KUKA KRL program: f1_Kuka_APT204T02S04.SRC

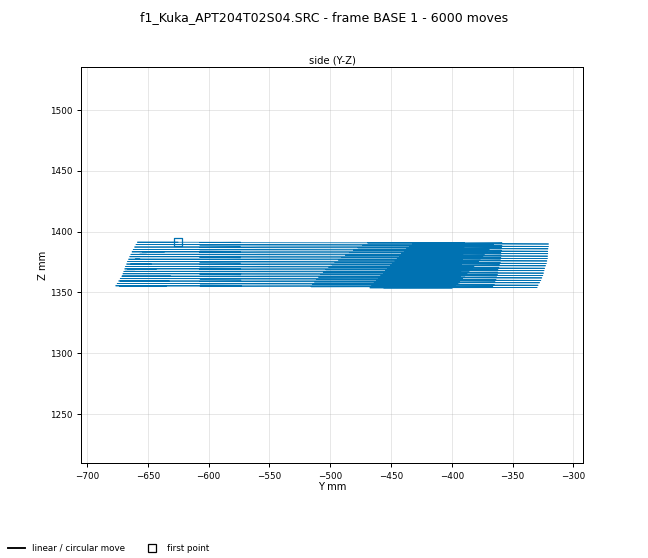
[picture p0: tool path of f1_Kuka_APT204T02S04.SRC in frame BASE 1, 6000 of 6001 moves have a stored position in this frame; points joined in program order, loops and branches not executed]
&ACCESS RVP
&REL 2
&PARAM TEMPLATE = C:\KRC\Roboter\Template\vorgabe
&PARAM EDITMASK = *
DEF f1_Kuka_APT204T02S04()


;FOLD INI;%{PE}%V3.2.0,%MKUKATPBASIS,%CINIT,%VCOMMON,%P
  ;FOLD BAS INI;%{E}%V3.2.0,%MKUKATPBASIS,%CINIT,%VINIT,%P
    GLOBAL INTERRUPT DECL 3 WHEN $STOPMESS==TRUE DO IR_STOPM ( )
    INTERRUPT ON 3
    BAS (#INITMOV,0 )
  ;ENDFOLD (BAS INI)
  ;FOLD USER INI;%{E}%V3.2.0,%MKUKATPUSER,%CINIT,%VINIT,%P
    ;Make your modifications here
  ;ENDFOLD (USER INI)
;ENDFOLD (INI)


;*** Make Null PTP Move
  PTP $pos_act

;*** Auto Load The Correct TOOL Data
  $tool=tool_data[2]

;*** Auto Load The Correct BASE Data
  $base=base_data[1]

  $ADVANCE = 5

;*** Restate Last Velocity
MMPM(30000.0)
SetRPM(8000)
LIN {X -0.143,Y -625.196,Z 1391.416,A 0.000,B 0.000,C 90.000,E1 110.791} C_DIS
LIN {X -0.238,Y -629.866,Z 1391.413,A 0.000,B 0.000,C 90.000,E1 110.301} C_DIS
LIN {X 0.179,Y -634.129,Z 1391.410,A 0.000,B 0.000,C 90.000,E1 109.758} C_DIS
LIN {X 0.021,Y -638.848,Z 1391.406,A 0.000,B 0.000,C 90.000,E1 109.141} C_DIS
LIN {X -0.310,Y -643.103,Z 1391.403,A 0.000,B 0.000,C 90.000,E1 108.544} C_DIS
LIN {X 0.208,Y -646.821,Z 1391.399,A 0.000,B 0.000,C 90.000,E1 107.873} C_DIS
LIN {X -0.083,Y -649.386,Z 1391.397,A 0.000,B 0.000,C 90.000,E1 107.402} C_DIS
LIN {X -0.030,Y -650.571,Z 1391.395,A 0.000,B 0.000,C 90.000,E1 107.149} C_DIS
LIN {X -0.300,Y -652.600,Z 1391.393,A 0.000,B 0.000,C 90.000,E1 106.677} C_DIS
LIN {X 0.197,Y -653.441,Z 1391.391,A 0.000,B 0.000,C 90.000,E1 106.386} C_DIS
LIN {X 0.134,Y -654.835,Z 1391.388,A 0.000,B 0.000,C 90.000,E1 105.898} C_DIS
LIN {X -0.217,Y -656.248,Z 1391.384,A 0.000,B 0.000,C 90.000,E1 105.190} C_DIS
LIN {X 0.139,Y -657.684,Z 1391.379,A 0.000,B 0.000,C 90.000,E1 104.175} C_DIS
LIN {X -0.185,Y -658.387,Z 1391.375,A 0.000,B 0.000,C 90.000,E1 103.467} C_DIS
LIN {X 0.242,Y -658.599,Z 1391.372,A 0.000,B 0.000,C 90.000,E1 102.939} C_DIS
LIN {X -0.216,Y -658.574,Z 1391.368,A 0.000,B 0.000,C 90.000,E1 102.243} C_DIS
LIN {X 0.219,Y -658.347,Z 1391.365,A 0.000,B 0.000,C 90.000,E1 101.715} C_DIS
LIN {X 0.004,Y -657.844,Z 1391.363,A 0.000,B 0.000,C 90.000,E1 101.243} C_DIS
LIN {X -0.340,Y -657.164,Z 1391.360,A 0.000,B 0.000,C 90.000,E1 100.782} C_DIS
LIN {X -0.034,Y -655.750,Z 1391.356,A 0.000,B 0.000,C 90.000,E1 100.018} C_DIS
LIN {X 0.261,Y -654.606,Z 1391.353,A 0.000,B 0.000,C 90.000,E1 99.500} C_DIS
LIN {X 0.012,Y -653.243,Z 1391.350,A 0.000,B 0.000,C 90.000,E1 99.029} C_DIS
LIN {X 0.158,Y -650.750,Z 1391.346,A 0.000,B 0.000,C 90.000,E1 98.276} C_DIS
LIN {X -0.217,Y -648.856,Z 1391.343,A 0.000,B 0.000,C 90.000,E1 97.814} C_DIS
LIN {X -0.196,Y -645.464,Z 1391.339,A 0.000,B 0.000,C 90.000,E1 97.068} C_DIS
LIN {X 0.043,Y -642.991,Z 1391.336,A 0.000,B 0.000,C 90.000,E1 96.549} C_DIS
LIN {X 0.261,Y -640.303,Z 1391.334,A 0.000,B 0.000,C 90.000,E1 96.030} C_DIS
LIN {X 0.262,Y -635.979,Z 1391.329,A 0.000,B 0.000,C 90.000,E1 95.277} C_DIS
LIN {X 0.290,Y -632.062,Z 1391.326,A 0.000,B 0.000,C 90.000,E1 94.645} C_DIS
LIN {X 0.283,Y -627.598,Z 1391.323,A 0.000,B 0.000,C 90.000,E1 94.012} C_DIS
LIN {X -0.280,Y -623.386,Z 1391.320,A 0.000,B 0.000,C 90.000,E1 93.555} C_DIS
LIN {X -0.233,Y -617.142,Z 1391.316,A 0.000,B 0.000,C 90.000,E1 92.922} C_DIS
LIN {X 0.002,Y -609.127,Z 1391.312,A 0.000,B 0.000,C 90.000,E1 92.178} C_DIS
LIN {X -0.133,Y -602.258,Z 1391.309,A 0.000,B 0.000,C 90.000,E1 91.604} C_DIS
LIN {X -0.057,Y -596.480,Z 1391.306,A 0.000,B 0.000,C 90.000,E1 91.146} C_DIS
LIN {X -0.147,Y -589.887,Z 1391.304,A 0.000,B 0.000,C 90.000,E1 90.745} C_DIS
LIN {X -0.112,Y -577.492,Z 1391.301,A 0.000,B 0.000,C 90.000,E1 90.115} C_DIS
LIN {X 0.014,Y -574.202,Z 1391.299,A 0.000,B 0.000,C 90.000,E1 89.771} C_DIS
LIN {X -0.190,Y -573.788,Z 1391.298,A 0.000,B 0.000,C 90.000,E1 89.599} C_DIS
LIN {X -0.045,Y -573.564,Z 1391.296,A 0.000,B 0.000,C 90.000,E1 89.312} C_DIS
LIN {X 0.026,Y -573.965,Z 1391.292,A 0.000,B 0.000,C 90.000,E1 88.625} C_DIS
LIN {X 0.192,Y -575.130,Z 1391.285,A 0.000,B 0.000,C 90.000,E1 87.249} C_DIS
LIN {X -0.193,Y -578.267,Z 1391.267,A 0.000,B 0.000,C 90.000,E1 84.033} C_DIS
LIN {X -0.072,Y -580.429,Z 1391.256,A 0.000,B 0.000,C 90.000,E1 82.129} C_DIS
LIN {X -0.185,Y -582.040,Z 1391.249,A 0.000,B 0.000,C 90.000,E1 80.792} C_DIS
LIN {X -0.262,Y -583.597,Z 1391.241,A 0.000,B 0.000,C 90.000,E1 79.454} C_DIS
LIN {X -0.202,Y -585.007,Z 1391.234,A 0.000,B 0.000,C 90.000,E1 78.105} C_DIS
LIN {X 0.135,Y -586.366,Z 1391.225,A 0.000,B 0.000,C 90.000,E1 76.464} C_DIS
LIN {X -0.014,Y -587.239,Z 1391.219,A 0.000,B 0.000,C 90.000,E1 75.408} C_DIS
LIN {X -0.008,Y -588.007,Z 1391.213,A 0.000,B 0.000,C 90.000,E1 74.338} C_DIS
LIN {X 0.104,Y -588.860,Z 1391.204,A 0.000,B 0.000,C 90.000,E1 72.725} C_DIS
LIN {X -0.146,Y -589.785,Z 1391.195,A 0.000,B 0.000,C 90.000,E1 71.148} C_DIS
LIN {X -0.253,Y -590.554,Z 1391.188,A 0.000,B 0.000,C 90.000,E1 69.826} C_DIS
LIN {X 0.057,Y -591.813,Z 1391.176,A 0.000,B 0.000,C 90.000,E1 67.667} C_DIS
LIN {X 0.193,Y -593.164,Z 1391.166,A 0.000,B 0.000,C 90.000,E1 65.793} C_DIS
LIN {X -0.016,Y -594.849,Z 1391.154,A 0.000,B 0.000,C 90.000,E1 63.691} C_DIS
LIN {X 0.160,Y -595.718,Z 1391.148,A 0.000,B 0.000,C 90.000,E1 62.615} C_DIS
LIN {X -0.128,Y -597.967,Z 1391.133,A 0.000,B 0.000,C 90.000,E1 59.999} C_DIS
LIN {X 0.200,Y -599.678,Z 1391.123,A 0.000,B 0.000,C 90.000,E1 58.122} C_DIS
LIN {X 0.057,Y -601.389,Z 1391.113,A 0.000,B 0.000,C 90.000,E1 56.294} C_DIS
LIN {X -0.219,Y -603.022,Z 1391.103,A 0.000,B 0.000,C 90.000,E1 54.482} C_DIS
LIN {X -0.002,Y -604.422,Z 1391.094,A 0.000,B 0.000,C 90.000,E1 52.889} C_DIS
LIN {X 0.200,Y -605.213,Z 1391.088,A 0.000,B 0.000,C 90.000,E1 51.823} C_DIS
LIN {X -0.070,Y -605.930,Z 1391.082,A 0.000,B 0.000,C 90.000,E1 50.803} C_DIS
LIN {X 0.119,Y -606.746,Z 1391.074,A 0.000,B 0.000,C 90.000,E1 49.218} C_DIS
LIN {X 0.062,Y -607.082,Z 1391.066,A 0.000,B 0.000,C 90.000,E1 47.919} C_DIS
LIN {X 0.003,Y -607.334,Z 1391.059,A 0.000,B 0.000,C 90.000,E1 46.620} C_DIS
LIN {X 0.297,Y -607.326,Z 1391.055,A 0.000,B 0.000,C 90.000,E1 45.810} C_DIS
LIN {X -0.025,Y -607.212,Z 1391.049,A 0.000,B 0.000,C 90.000,E1 44.798} C_DIS
LIN {X -0.096,Y -606.832,Z 1391.042,A 0.000,B 0.000,C 90.000,E1 43.500} C_DIS
LIN {X 0.001,Y -606.333,Z 1391.036,A 0.000,B 0.000,C 90.000,E1 42.447} C_DIS
LIN {X -0.133,Y -605.921,Z 1391.031,A 0.000,B 0.000,C 90.000,E1 41.676} C_DIS
LIN {X -0.214,Y -605.096,Z 1391.024,A 0.000,B 0.000,C 90.000,E1 40.378} C_DIS
LIN {X 0.148,Y -604.051,Z 1391.017,A 0.000,B 0.000,C 90.000,E1 39.036} C_DIS
LIN {X 0.112,Y -602.680,Z 1391.010,A 0.000,B 0.000,C 90.000,E1 37.729} C_DIS
LIN {X 0.030,Y -601.770,Z 1391.005,A 0.000,B 0.000,C 90.000,E1 36.950} C_DIS
LIN {X 0.191,Y -600.161,Z 1391.000,A 0.000,B 0.000,C 90.000,E1 35.884} C_DIS
LIN {X 0.087,Y -598.794,Z 1390.995,A 0.000,B 0.000,C 90.000,E1 35.105} C_DIS
LIN {X -0.033,Y -597.155,Z 1390.991,A 0.000,B 0.000,C 90.000,E1 34.326} C_DIS
LIN {X -0.064,Y -594.161,Z 1390.983,A 0.000,B 0.000,C 90.000,E1 33.007} C_DIS
LIN {X -0.065,Y -592.043,Z 1390.979,A 0.000,B 0.000,C 90.000,E1 32.212} C_DIS
LIN {X -0.080,Y -589.699,Z 1390.974,A 0.000,B 0.000,C 90.000,E1 31.416} C_DIS
LIN {X 0.114,Y -588.884,Z 1390.973,A 0.000,B 0.000,C 90.000,E1 31.131} C_DIS
LIN {X 0.066,Y -586.005,Z 1390.969,A 0.000,B 0.000,C 90.000,E1 30.335} C_DIS
LIN {X -0.011,Y -582.750,Z 1390.964,A 0.000,B 0.000,C 90.000,E1 29.539} C_DIS
LIN {X -0.191,Y -578.488,Z 1390.959,A 0.000,B 0.000,C 90.000,E1 28.615} C_DIS
LIN {X 0.031,Y -575.870,Z 1390.956,A 0.000,B 0.000,C 90.000,E1 28.052} C_DIS
LIN {X -0.003,Y -573.037,Z 1390.953,A 0.000,B 0.000,C 90.000,E1 27.513} C_DIS
LIN {X -0.067,Y -567.662,Z 1390.948,A 0.000,B 0.000,C 90.000,E1 26.565} C_DIS
LIN {X 0.243,Y -563.612,Z 1390.944,A 0.000,B 0.000,C 90.000,E1 25.848} C_DIS
LIN {X -0.139,Y -560.160,Z 1390.941,A 0.000,B 0.000,C 90.000,E1 25.335} C_DIS
LIN {X -0.038,Y -556.507,Z 1390.938,A 0.000,B 0.000,C 90.000,E1 24.771} C_DIS
LIN {X -0.073,Y -551.522,Z 1390.934,A 0.000,B 0.000,C 90.000,E1 24.079} C_DIS
LIN {X 0.085,Y -548.354,Z 1390.931,A 0.000,B 0.000,C 90.000,E1 23.643} C_DIS
LIN {X 0.103,Y -542.913,Z 1390.928,A 0.000,B 0.000,C 90.000,E1 22.950} C_DIS
LIN {X -0.059,Y -537.032,Z 1390.924,A 0.000,B 0.000,C 90.000,E1 22.259} C_DIS
LIN {X -0.231,Y -528.146,Z 1390.918,A 0.000,B 0.000,C 90.000,E1 21.280} C_DIS
LIN {X -0.094,Y -521.657,Z 1390.914,A 0.000,B 0.000,C 90.000,E1 20.556} C_DIS
LIN {X -0.150,Y -512.419,Z 1390.909,A 0.000,B 0.000,C 90.000,E1 19.577} C_DIS
LIN {X -0.058,Y -501.874,Z 1390.903,A 0.000,B 0.000,C 90.000,E1 18.489} C_DIS
LIN {X -0.108,Y -486.810,Z 1390.894,A 0.000,B 0.000,C 90.000,E1 16.968} C_DIS
LIN {X 0.057,Y -471.479,Z 1390.885,A 0.000,B 0.000,C 90.000,E1 15.371} C_DIS
LIN {X -0.025,Y -461.668,Z 1390.880,A 0.000,B 0.000,C 90.000,E1 14.356} C_DIS
LIN {X 0.031,Y -447.810,Z 1390.872,A 0.000,B 0.000,C 90.000,E1 12.883} C_DIS
LIN {X -0.238,Y -428.554,Z 1390.860,A 0.000,B 0.000,C 90.000,E1 10.782} C_DIS
LIN {X -0.101,Y -410.782,Z 1390.848,A 0.000,B 0.000,C 90.000,E1 8.624} C_DIS
LIN {X 0.175,Y -396.943,Z 1390.839,A 0.000,B 0.000,C 90.000,E1 6.891} C_DIS
LIN {X 0.154,Y -392.878,Z 1390.836,A 0.000,B 0.000,C 90.000,E1 6.372} C_DIS
LIN {X 0.048,Y -389.976,Z 1390.833,A 0.000,B 0.000,C 90.000,E1 5.910} C_DIS
LIN {X 0.011,Y -389.942,Z 1390.833,A 0.000,B 0.000,C 90.000,E1 5.910} C_DIS
LIN {X -0.120,Y -389.697,Z 1390.832,A 0.000,B 0.000,C 90.000,E1 5.796} C_DIS
LIN {X -0.158,Y -389.698,Z 1390.832,A 0.000,B 0.000,C 90.000,E1 5.796} C_DIS
LIN {X -0.089,Y -390.823,Z 1390.831,A 0.000,B 0.000,C 90.000,E1 5.625} C_DIS
LIN {X 0.121,Y -393.551,Z 1390.829,A 0.000,B 0.000,C 90.000,E1 5.277} C_DIS
LIN {X 0.038,Y -404.905,Z 1390.824,A 0.000,B 0.000,C 90.000,E1 4.302} C_DIS
LIN {X -0.100,Y -409.448,Z 1390.822,A 0.000,B 0.000,C 90.000,E1 3.898} C_DIS
LIN {X -0.163,Y -412.171,Z 1390.820,A 0.000,B 0.000,C 90.000,E1 3.612} C_DIS
LIN {X -0.101,Y -417.094,Z 1390.817,A 0.000,B 0.000,C 90.000,E1 3.037} C_DIS
LIN {X 0.084,Y -423.352,Z 1390.812,A 0.000,B 0.000,C 90.000,E1 2.178} C_DIS
LIN {X 0.192,Y -427.973,Z 1390.808,A 0.000,B 0.000,C 90.000,E1 1.489} C_DIS
LIN {X -0.107,Y -432.450,Z 1390.805,A 0.000,B 0.000,C 90.000,E1 0.859} C_DIS
LIN {X 0.000,Y -437.845,Z 1390.800,A 0.000,B 0.000,C 90.000,E1 360.000} C_DIS
LIN {X -0.049,Y -443.155,Z 1390.795,A 0.000,B 0.000,C 90.000,E1 359.141} C_DIS
LIN {X 0.209,Y -447.035,Z 1390.792,A 0.000,B 0.000,C 90.000,E1 358.453} C_DIS
LIN {X 0.222,Y -452.233,Z 1390.786,A 0.000,B 0.000,C 90.000,E1 357.478} C_DIS
LIN {X 0.212,Y -456.335,Z 1390.782,A 0.000,B 0.000,C 90.000,E1 356.674} C_DIS
LIN {X 0.118,Y -459.401,Z 1390.778,A 0.000,B 0.000,C 90.000,E1 356.045} C_DIS
LIN {X -0.150,Y -463.497,Z 1390.773,A 0.000,B 0.000,C 90.000,E1 355.122} C_DIS
LIN {X 0.156,Y -465.457,Z 1390.770,A 0.000,B 0.000,C 90.000,E1 354.609} C_DIS
LIN {X 0.156,Y -467.659,Z 1390.767,A 0.000,B 0.000,C 90.000,E1 353.976} C_DIS
LIN {X -0.044,Y -468.494,Z 1390.765,A 0.000,B 0.000,C 90.000,E1 353.685} C_DIS
LIN {X 0.225,Y -469.028,Z 1390.763,A 0.000,B 0.000,C 90.000,E1 353.337} C_DIS
LIN {X -0.023,Y -469.181,Z 1390.761,A 0.000,B 0.000,C 90.000,E1 353.053} C_DIS
LIN {X -0.211,Y -468.449,Z 1390.760,A 0.000,B 0.000,C 90.000,E1 352.761} C_DIS
LIN {X -0.022,Y -467.671,Z 1390.759,A 0.000,B 0.000,C 90.000,E1 352.648} C_DIS
LIN {X -0.135,Y -465.013,Z 1390.759,A 0.000,B 0.000,C 90.000,E1 352.591} C_DIS
LIN {X -0.105,Y -421.785,Z 1390.755,A 0.000,B 0.000,C 90.000,E1 351.837} C_DIS
LIN {X 0.169,Y -384.990,Z 1390.750,A 0.000,B 0.000,C 90.000,E1 351.027} C_DIS
LIN {X 0.119,Y -358.693,Z 1390.747,A 0.000,B 0.000,C 90.000,E1 350.387} C_DIS
LIN {X 0.100,Y -358.666,Z 1390.747,A 0.000,B 0.000,C 90.000,E1 350.387} C_DIS
LIN {X -0.096,Y -359.584,Z 1390.725,A 0.000,B 0.000,C 90.000,E1 346.589} C_DIS
LIN {X -0.088,Y -361.850,Z 1390.684,A 0.000,B 0.000,C 90.000,E1 339.082} C_DIS
LIN {X 0.207,Y -362.253,Z 1390.675,A 0.000,B 0.000,C 90.000,E1 337.539} C_DIS
LIN {X 0.082,Y -366.046,Z 1390.642,A 0.000,B 0.000,C 90.000,E1 331.591} C_DIS
LIN {X -0.212,Y -367.179,Z 1390.630,A 0.000,B 0.000,C 90.000,E1 329.410} C_DIS
LIN {X 0.044,Y -371.805,Z 1390.601,A 0.000,B 0.000,C 90.000,E1 324.196} C_DIS
LIN {X -0.168,Y -377.442,Z 1390.567,A 0.000,B 0.000,C 90.000,E1 318.000} C_DIS
LIN {X 0.112,Y -378.276,Z 1390.563,A 0.000,B 0.000,C 90.000,E1 317.229} C_DIS
LIN {X 0.108,Y -384.028,Z 1390.530,A 0.000,B 0.000,C 90.000,E1 311.434} C_DIS
LIN {X 0.194,Y -384.936,Z 1390.526,A 0.000,B 0.000,C 90.000,E1 310.701} C_DIS
LIN {X -0.177,Y -390.698,Z 1390.495,A 0.000,B 0.000,C 90.000,E1 305.025} C_DIS
LIN {X 0.210,Y -391.195,Z 1390.493,A 0.000,B 0.000,C 90.000,E1 304.612} C_DIS
LIN {X 0.017,Y -396.910,Z 1390.459,A 0.000,B 0.000,C 90.000,E1 298.615} C_DIS
LIN {X -0.109,Y -397.907,Z 1390.449,A 0.000,B 0.000,C 90.000,E1 296.873} C_DIS
LIN {X 0.028,Y -401.639,Z 1390.426,A 0.000,B 0.000,C 90.000,E1 292.642} C_DIS
LIN {X 0.165,Y -404.713,Z 1390.395,A 0.000,B 0.000,C 90.000,E1 287.040} C_DIS
LIN {X 0.168,Y -406.136,Z 1390.364,A 0.000,B 0.000,C 90.000,E1 281.478} C_DIS
LIN {X -0.135,Y -405.443,Z 1390.347,A 0.000,B 0.000,C 90.000,E1 278.398} C_DIS
LIN {X -0.138,Y -405.689,Z 1390.333,A 0.000,B 0.000,C 90.000,E1 275.967} C_DIS
LIN {X -0.067,Y -403.574,Z 1390.306,A 0.000,B 0.000,C 90.000,E1 271.088} C_DIS
LIN {X -0.132,Y -403.240,Z 1390.302,A 0.000,B 0.000,C 90.000,E1 270.401} C_DIS
LIN {X 0.106,Y -399.091,Z 1390.273,A 0.000,B 0.000,C 90.000,E1 265.122} C_DIS
LIN {X 0.048,Y -398.855,Z 1390.271,A 0.000,B 0.000,C 90.000,E1 264.780} C_DIS
LIN {X -0.054,Y -393.336,Z 1390.244,A 0.000,B 0.000,C 90.000,E1 259.859} C_DIS
LIN {X -0.133,Y -392.758,Z 1390.240,A 0.000,B 0.000,C 90.000,E1 259.162} C_DIS
LIN {X -0.054,Y -386.308,Z 1390.214,A 0.000,B 0.000,C 90.000,E1 254.519} C_DIS
LIN {X 0.018,Y -385.205,Z 1390.208,A 0.000,B 0.000,C 90.000,E1 253.433} C_DIS
LIN {X -0.051,Y -383.992,Z 1390.204,A 0.000,B 0.000,C 90.000,E1 252.725} C_DIS
LIN {X -0.221,Y -377.431,Z 1390.180,A 0.000,B 0.000,C 90.000,E1 248.411} C_DIS
LIN {X 0.016,Y -376.161,Z 1390.174,A 0.000,B 0.000,C 90.000,E1 247.283} C_DIS
LIN {X 0.187,Y -368.327,Z 1390.147,A 0.000,B 0.000,C 90.000,E1 242.487} C_DIS
LIN {X -0.097,Y -366.466,Z 1390.139,A 0.000,B 0.000,C 90.000,E1 241.051} C_DIS
LIN {X -0.012,Y -365.918,Z 1390.137,A 0.000,B 0.000,C 90.000,E1 240.667} C_DIS
LIN {X 0.077,Y -359.101,Z 1390.114,A 0.000,B 0.000,C 90.000,E1 236.548} C_DIS
LIN {X 0.164,Y -356.245,Z 1390.102,A 0.000,B 0.000,C 90.000,E1 234.276} C_DIS
LIN {X 0.095,Y -355.717,Z 1390.100,A 0.000,B 0.000,C 90.000,E1 233.909} C_DIS
LIN {X -0.101,Y -348.706,Z 1390.074,A 0.000,B 0.000,C 90.000,E1 229.380} C_DIS
LIN {X -0.027,Y -346.116,Z 1390.062,A 0.000,B 0.000,C 90.000,E1 227.067} C_DIS
LIN {X -0.041,Y -342.667,Z 1390.049,A 0.000,B 0.000,C 90.000,E1 224.757} C_DIS
LIN {X 0.152,Y -336.754,Z 1390.018,A 0.000,B 0.000,C 90.000,E1 219.277} C_DIS
LIN {X 0.062,Y -330.806,Z 1389.988,A 0.000,B 0.000,C 90.000,E1 213.785} C_DIS
LIN {X 0.019,Y -329.252,Z 1389.975,A 0.000,B 0.000,C 90.000,E1 211.416} C_DIS
LIN {X -0.130,Y -324.635,Z 1389.941,A 0.000,B 0.000,C 90.000,E1 205.463} C_DIS
LIN {X 0.062,Y -323.806,Z 1389.928,A 0.000,B 0.000,C 90.000,E1 203.025} C_DIS
LIN {X -0.034,Y -321.131,Z 1389.881,A 0.000,B 0.000,C 90.000,E1 194.592} C_DIS
LIN {X -0.062,Y -320.418,Z 1389.862,A 0.000,B 0.000,C 90.000,E1 191.243} C_DIS
LIN {X -0.092,Y -320.565,Z 1389.862,A 0.000,B 0.000,C 90.000,E1 191.243} C_DIS
LIN {X 0.115,Y -350.932,Z 1389.857,A 0.000,B 0.000,C 90.000,E1 190.254} C_DIS
LIN {X 0.078,Y -384.592,Z 1389.852,A 0.000,B 0.000,C 90.000,E1 189.378} C_DIS
LIN {X 0.108,Y -424.277,Z 1389.847,A 0.000,B 0.000,C 90.000,E1 188.511} C_DIS
LIN {X 0.124,Y -429.421,Z 1389.847,A 0.000,B 0.000,C 90.000,E1 188.398} C_DIS
LIN {X -0.080,Y -430.370,Z 1389.846,A 0.000,B 0.000,C 90.000,E1 188.341} C_DIS
LIN {X 0.070,Y -431.572,Z 1389.845,A 0.000,B 0.000,C 90.000,E1 188.049} C_DIS
LIN {X 0.182,Y -432.160,Z 1389.843,A 0.000,B 0.000,C 90.000,E1 187.701} C_DIS
LIN {X -0.131,Y -432.366,Z 1389.841,A 0.000,B 0.000,C 90.000,E1 187.409} C_DIS
LIN {X 0.051,Y -432.032,Z 1389.837,A 0.000,B 0.000,C 90.000,E1 186.720} C_DIS
LIN {X 0.030,Y -431.325,Z 1389.830,A 0.000,B 0.000,C 90.000,E1 185.391} C_DIS
LIN {X -0.152,Y -430.337,Z 1389.824,A 0.000,B 0.000,C 90.000,E1 184.416} C_DIS
LIN {X 0.018,Y -429.583,Z 1389.821,A 0.000,B 0.000,C 90.000,E1 183.726} C_DIS
LIN {X -0.114,Y -427.646,Z 1389.813,A 0.000,B 0.000,C 90.000,E1 182.407} C_DIS
LIN {X 0.029,Y -426.466,Z 1389.810,A 0.000,B 0.000,C 90.000,E1 181.718} C_DIS
LIN {X 0.205,Y -424.428,Z 1389.804,A 0.000,B 0.000,C 90.000,E1 180.688} C_DIS
LIN {X -0.165,Y -423.680,Z 1389.802,A 0.000,B 0.000,C 90.000,E1 180.401} C_DIS
LIN {X -0.019,Y -420.873,Z 1389.797,A 0.000,B 0.000,C 90.000,E1 179.370} C_DIS
LIN {X 0.057,Y -418.810,Z 1389.793,A 0.000,B 0.000,C 90.000,E1 178.682} C_DIS
LIN {X 0.148,Y -415.012,Z 1389.787,A 0.000,B 0.000,C 90.000,E1 177.650} C_DIS
LIN {X 0.191,Y -411.516,Z 1389.782,A 0.000,B 0.000,C 90.000,E1 176.788} C_DIS
LIN {X 0.190,Y -406.155,Z 1389.777,A 0.000,B 0.000,C 90.000,E1 175.755} C_DIS
LIN {X 0.141,Y -401.143,Z 1389.772,A 0.000,B 0.000,C 90.000,E1 174.894} C_DIS
LIN {X -0.127,Y -387.572,Z 1389.760,A 0.000,B 0.000,C 90.000,E1 172.818} C_DIS
LIN {X -0.015,Y -380.337,Z 1389.753,A 0.000,B 0.000,C 90.000,E1 171.546} C_DIS
LIN {X -0.033,Y -372.669,Z 1389.745,A 0.000,B 0.000,C 90.000,E1 170.095} C_DIS
LIN {X 0.090,Y -369.184,Z 1389.741,A 0.000,B 0.000,C 90.000,E1 169.342} C_DIS
LIN {X 0.017,Y -367.117,Z 1389.738,A 0.000,B 0.000,C 90.000,E1 168.814} C_DIS
LIN {X 0.005,Y -365.770,Z 1389.735,A 0.000,B 0.000,C 90.000,E1 168.285} C_DIS
LIN {X -0.032,Y -365.767,Z 1389.735,A 0.000,B 0.000,C 90.000,E1 168.285} C_DIS
LIN {X 0.093,Y -366.445,Z 1389.733,A 0.000,B 0.000,C 90.000,E1 167.825} C_DIS
LIN {X 0.056,Y -366.477,Z 1389.732,A 0.000,B 0.000,C 90.000,E1 167.825} C_DIS
LIN {X -0.040,Y -369.073,Z 1389.730,A 0.000,B 0.000,C 90.000,E1 167.353} C_DIS
LIN {X 0.057,Y -376.139,Z 1389.725,A 0.000,B 0.000,C 90.000,E1 166.408} C_DIS
LIN {X -0.008,Y -383.314,Z 1389.720,A 0.000,B 0.000,C 90.000,E1 165.589} C_DIS
LIN {X -0.071,Y -395.482,Z 1389.713,A 0.000,B 0.000,C 90.000,E1 164.338} C_DIS
LIN {X 0.143,Y -407.819,Z 1389.707,A 0.000,B 0.000,C 90.000,E1 163.142} C_DIS
LIN {X -0.231,Y -431.267,Z 1389.696,A 0.000,B 0.000,C 90.000,E1 161.221} C_DIS
LIN {X 0.064,Y -443.907,Z 1389.690,A 0.000,B 0.000,C 90.000,E1 160.188} C_DIS
LIN {X -0.031,Y -454.875,Z 1389.685,A 0.000,B 0.000,C 90.000,E1 159.337} C_DIS
LIN {X -0.012,Y -465.637,Z 1389.680,A 0.000,B 0.000,C 90.000,E1 158.465} C_DIS
LIN {X -0.180,Y -473.094,Z 1389.677,A 0.000,B 0.000,C 90.000,E1 157.847} C_DIS
LIN {X -0.046,Y -478.923,Z 1389.674,A 0.000,B 0.000,C 90.000,E1 157.305} C_DIS
LIN {X -0.136,Y -487.315,Z 1389.670,A 0.000,B 0.000,C 90.000,E1 156.538} C_DIS
LIN {X -0.108,Y -494.325,Z 1389.666,A 0.000,B 0.000,C 90.000,E1 155.869} C_DIS
LIN {X -0.040,Y -502.435,Z 1389.661,A 0.000,B 0.000,C 90.000,E1 155.025} C_DIS
LIN {X -0.105,Y -507.695,Z 1389.658,A 0.000,B 0.000,C 90.000,E1 154.460} C_DIS
LIN {X -0.048,Y -514.044,Z 1389.654,A 0.000,B 0.000,C 90.000,E1 153.717} C_DIS
LIN {X -0.213,Y -519.975,Z 1389.650,A 0.000,B 0.000,C 90.000,E1 152.999} C_DIS
LIN {X -0.005,Y -523.355,Z 1389.647,A 0.000,B 0.000,C 90.000,E1 152.538} C_DIS
LIN {X -0.022,Y -526.518,Z 1389.645,A 0.000,B 0.000,C 90.000,E1 152.103} C_DIS
LIN {X 0.074,Y -530.265,Z 1389.642,A 0.000,B 0.000,C 90.000,E1 151.513} C_DIS
LIN {X 0.055,Y -534.335,Z 1389.638,A 0.000,B 0.000,C 90.000,E1 150.795} C_DIS
LIN {X 0.210,Y -537.186,Z 1389.635,A 0.000,B 0.000,C 90.000,E1 150.205} C_DIS
LIN {X -0.220,Y -540.124,Z 1389.631,A 0.000,B 0.000,C 90.000,E1 149.537} C_DIS
LIN {X -0.028,Y -542.270,Z 1389.628,A 0.000,B 0.000,C 90.000,E1 148.948} C_DIS
LIN {X 0.195,Y -545.040,Z 1389.623,A 0.000,B 0.000,C 90.000,E1 148.074} C_DIS
LIN {X -0.041,Y -546.655,Z 1389.620,A 0.000,B 0.000,C 90.000,E1 147.533} C_DIS
LIN {X -0.230,Y -548.631,Z 1389.615,A 0.000,B 0.000,C 90.000,E1 146.707} C_DIS
LIN {X 0.368,Y -550.363,Z 1389.610,A 0.000,B 0.000,C 90.000,E1 145.801} C_DIS
LIN {X 0.222,Y -551.768,Z 1389.606,A 0.000,B 0.000,C 90.000,E1 144.975} C_DIS
LIN {X 0.086,Y -552.876,Z 1389.601,A 0.000,B 0.000,C 90.000,E1 144.149} C_DIS
LIN {X -0.094,Y -553.976,Z 1389.595,A 0.000,B 0.000,C 90.000,E1 143.050} C_DIS
LIN {X -0.097,Y -555.317,Z 1389.585,A 0.000,B 0.000,C 90.000,E1 141.376} C_DIS
LIN {X -0.155,Y -556.399,Z 1389.578,A 0.000,B 0.000,C 90.000,E1 139.989} C_DIS
LIN {X 0.007,Y -556.905,Z 1389.573,A 0.000,B 0.000,C 90.000,E1 139.138} C_DIS
LIN {X -0.088,Y -557.589,Z 1389.565,A 0.000,B 0.000,C 90.000,E1 137.757} C_DIS
LIN {X -0.065,Y -558.334,Z 1389.555,A 0.000,B 0.000,C 90.000,E1 135.810} C_DIS
LIN {X -0.162,Y -558.860,Z 1389.547,A 0.000,B 0.000,C 90.000,E1 134.433} C_DIS
LIN {X -0.183,Y -559.391,Z 1389.538,A 0.000,B 0.000,C 90.000,E1 132.771} C_DIS
LIN {X 0.214,Y -559.667,Z 1389.528,A 0.000,B 0.000,C 90.000,E1 131.067} C_DIS
LIN {X -0.022,Y -560.050,Z 1389.518,A 0.000,B 0.000,C 90.000,E1 129.152} C_DIS
LIN {X -0.243,Y -560.611,Z 1389.507,A 0.000,B 0.000,C 90.000,E1 127.237} C_DIS
LIN {X 0.238,Y -561.334,Z 1389.499,A 0.000,B 0.000,C 90.000,E1 125.804} C_DIS
LIN {X -0.005,Y -561.741,Z 1389.497,A 0.000,B 0.000,C 90.000,E1 125.518} C_DIS
LIN {X -0.352,Y -562.723,Z 1389.496,A 0.000,B 0.000,C 90.000,E1 125.311} C_DIS
LIN {X 0.082,Y -563.387,Z 1389.494,A 0.000,B 0.000,C 90.000,E1 124.978} C_DIS
LIN {X 0.039,Y -563.430,Z 1389.494,A 0.000,B 0.000,C 90.000,E1 124.978} C_DIS
LIN {X -0.041,Y -565.054,Z 1389.494,A 0.000,B 0.000,C 90.000,E1 124.865} C_DIS
LIN {X -0.259,Y -566.721,Z 1389.493,A 0.000,B 0.000,C 90.000,E1 124.818} C_DIS
LIN {X -0.196,Y -570.932,Z 1389.493,A 0.000,B 0.000,C 90.000,E1 124.692} C_DIS
LIN {X 0.099,Y -576.932,Z 1389.492,A 0.000,B 0.000,C 90.000,E1 124.532} C_DIS
LIN {X 0.090,Y -583.270,Z 1389.491,A 0.000,B 0.000,C 90.000,E1 124.358} C_DIS
LIN {X 0.074,Y -588.758,Z 1389.490,A 0.000,B 0.000,C 90.000,E1 124.119} C_DIS
LIN {X 0.168,Y -594.673,Z 1389.488,A 0.000,B 0.000,C 90.000,E1 123.785} C_DIS
LIN {X 0.059,Y -600.403,Z 1389.486,A 0.000,B 0.000,C 90.000,E1 123.420} C_DIS
LIN {X -0.015,Y -605.851,Z 1389.483,A 0.000,B 0.000,C 90.000,E1 123.007} C_DIS
LIN {X 0.199,Y -612.491,Z 1389.480,A 0.000,B 0.000,C 90.000,E1 122.418} C_DIS
LIN {X -0.116,Y -615.103,Z 1389.479,A 0.000,B 0.000,C 90.000,E1 122.212} C_DIS
LIN {X -0.069,Y -620.916,Z 1389.476,A 0.000,B 0.000,C 90.000,E1 121.592} C_DIS
LIN {X -0.090,Y -624.377,Z 1389.473,A 0.000,B 0.000,C 90.000,E1 121.209} C_DIS
LIN {X -0.285,Y -631.549,Z 1389.468,A 0.000,B 0.000,C 90.000,E1 120.335} C_DIS
LIN {X 0.105,Y -635.824,Z 1389.465,A 0.000,B 0.000,C 90.000,E1 119.667} C_DIS
LIN {X 0.195,Y -639.048,Z 1389.462,A 0.000,B 0.000,C 90.000,E1 119.155} C_DIS
LIN {X -0.220,Y -642.382,Z 1389.459,A 0.000,B 0.000,C 90.000,E1 118.565} C_DIS
LIN {X 0.152,Y -643.495,Z 1389.457,A 0.000,B 0.000,C 90.000,E1 118.281} C_DIS
LIN {X 0.294,Y -645.428,Z 1389.454,A 0.000,B 0.000,C 90.000,E1 117.769} C_DIS
LIN {X 0.371,Y -646.208,Z 1389.453,A 0.000,B 0.000,C 90.000,E1 117.513} C_DIS
LIN {X -0.041,Y -647.245,Z 1389.450,A 0.000,B 0.000,C 90.000,E1 117.052} C_DIS
LIN {X 0.043,Y -647.666,Z 1389.449,A 0.000,B 0.000,C 90.000,E1 116.796} C_DIS
LIN {X 0.129,Y -647.863,Z 1389.448,A 0.000,B 0.000,C 90.000,E1 116.539} C_DIS
LIN {X -0.072,Y -647.895,Z 1389.446,A 0.000,B 0.000,C 90.000,E1 116.309} C_DIS
LIN {X 0.198,Y -647.461,Z 1389.442,A 0.000,B 0.000,C 90.000,E1 115.540} C_DIS
LIN {X -0.212,Y -646.859,Z 1389.439,A 0.000,B 0.000,C 90.000,E1 115.079} C_DIS
LIN {X -0.128,Y -646.078,Z 1389.438,A 0.000,B 0.000,C 90.000,E1 114.823} C_DIS
LIN {X -0.232,Y -644.029,Z 1389.435,A 0.000,B 0.000,C 90.000,E1 114.335} C_DIS
LIN {X -0.084,Y -640.444,Z 1389.432,A 0.000,B 0.000,C 90.000,E1 113.823} C_DIS
LIN {X -0.053,Y -639.110,Z 1389.432,A 0.000,B 0.000,C 90.000,E1 113.695} C_DIS
LIN {X 0.212,Y -635.318,Z 1389.431,A 0.000,B 0.000,C 90.000,E1 113.462} C_DIS
LIN {X 0.116,Y -634.024,Z 1389.430,A 0.000,B 0.000,C 90.000,E1 113.387} C_DIS
LIN {X 0.270,Y -632.549,Z 1389.429,A 0.000,B 0.000,C 90.000,E1 113.259} C_DIS
LIN {X -0.344,Y -630.253,Z 1389.429,A 0.000,B 0.000,C 90.000,E1 113.206} C_DIS
LIN {X -0.112,Y -628.422,Z 1389.428,A 0.000,B 0.000,C 90.000,E1 113.131} C_DIS
LIN {X 0.252,Y -623.334,Z 1389.427,A 0.000,B 0.000,C 90.000,E1 112.898} C_DIS
LIN {X 0.292,Y -621.466,Z 1389.427,A 0.000,B 0.000,C 90.000,E1 112.823} C_DIS
LIN {X -0.010,Y -608.882,Z 1389.425,A 0.000,B 0.000,C 90.000,E1 112.461} C_DIS
LIN {X -0.043,Y -608.884,Z 1389.425,A 0.000,B 0.000,C 90.000,E1 112.461} C_DIS
LIN {X 0.139,Y -611.746,Z 1389.423,A 0.000,B 0.000,C 90.000,E1 112.153} C_DIS
LIN {X 0.064,Y -614.838,Z 1389.422,A 0.000,B 0.000,C 90.000,E1 111.897} C_DIS
LIN {X 0.306,Y -621.292,Z 1389.418,A 0.000,B 0.000,C 90.000,E1 111.280} C_DIS
LIN {X -0.243,Y -625.045,Z 1389.416,A 0.000,B 0.000,C 90.000,E1 110.972} C_DIS
LIN {X 0.285,Y -629.756,Z 1389.414,A 0.000,B 0.000,C 90.000,E1 110.429} C_DIS
LIN {X 0.113,Y -635.026,Z 1389.410,A 0.000,B 0.000,C 90.000,E1 109.812} C_DIS
LIN {X -0.249,Y -639.706,Z 1389.407,A 0.000,B 0.000,C 90.000,E1 109.214} C_DIS
LIN {X 0.243,Y -643.906,Z 1389.403,A 0.000,B 0.000,C 90.000,E1 108.544} C_DIS
LIN {X -0.042,Y -647.643,Z 1389.400,A 0.000,B 0.000,C 90.000,E1 107.946} C_DIS
LIN {X -0.104,Y -650.825,Z 1389.396,A 0.000,B 0.000,C 90.000,E1 107.330} C_DIS
LIN {X 0.126,Y -653.948,Z 1389.392,A 0.000,B 0.000,C 90.000,E1 106.567} C_DIS
LIN {X -0.050,Y -656.073,Z 1389.388,A 0.000,B 0.000,C 90.000,E1 105.843} C_DIS
LIN {X -0.388,Y -657.439,Z 1389.384,A 0.000,B 0.000,C 90.000,E1 105.134} C_DIS
LIN {X -0.013,Y -658.898,Z 1389.379,A 0.000,B 0.000,C 90.000,E1 104.120} C_DIS
LIN {X 0.316,Y -659.550,Z 1389.374,A 0.000,B 0.000,C 90.000,E1 103.355} C_DIS
LIN {X 0.113,Y -659.765,Z 1389.372,A 0.000,B 0.000,C 90.000,E1 102.883} C_DIS
LIN {X -0.193,Y -659.677,Z 1389.368,A 0.000,B 0.000,C 90.000,E1 102.175} C_DIS
LIN {X 0.111,Y -659.420,Z 1389.365,A 0.000,B 0.000,C 90.000,E1 101.658} C_DIS
LIN {X -0.096,Y -658.910,Z 1389.362,A 0.000,B 0.000,C 90.000,E1 101.186} C_DIS
LIN {X 0.338,Y -658.236,Z 1389.359,A 0.000,B 0.000,C 90.000,E1 100.658} C_DIS
LIN {X -0.114,Y -656.751,Z 1389.355,A 0.000,B 0.000,C 90.000,E1 99.962} C_DIS
LIN {X 0.190,Y -655.575,Z 1389.353,A 0.000,B 0.000,C 90.000,E1 99.443} C_DIS
LIN {X -0.052,Y -654.185,Z 1389.350,A 0.000,B 0.000,C 90.000,E1 98.973} C_DIS
LIN {X 0.239,Y -652.557,Z 1389.347,A 0.000,B 0.000,C 90.000,E1 98.454} C_DIS
LIN {X -0.124,Y -650.743,Z 1389.344,A 0.000,B 0.000,C 90.000,E1 97.992} C_DIS
LIN {X 0.001,Y -647.508,Z 1389.340,A 0.000,B 0.000,C 90.000,E1 97.239} C_DIS
LIN {X 0.132,Y -644.442,Z 1389.337,A 0.000,B 0.000,C 90.000,E1 96.606} C_DIS
LIN {X 0.305,Y -641.109,Z 1389.333,A 0.000,B 0.000,C 90.000,E1 95.967} C_DIS
LIN {X 0.247,Y -636.768,Z 1389.329,A 0.000,B 0.000,C 90.000,E1 95.220} C_DIS
LIN {X 0.282,Y -632.828,Z 1389.326,A 0.000,B 0.000,C 90.000,E1 94.588} C_DIS
LIN {X -0.254,Y -629.328,Z 1389.323,A 0.000,B 0.000,C 90.000,E1 94.131} C_DIS
LIN {X -0.277,Y -624.144,Z 1389.319,A 0.000,B 0.000,C 90.000,E1 93.498} C_DIS
LIN {X -0.225,Y -617.887,Z 1389.316,A 0.000,B 0.000,C 90.000,E1 92.865} C_DIS
LIN {X -0.013,Y -609.915,Z 1389.312,A 0.000,B 0.000,C 90.000,E1 92.121} C_DIS
LIN {X -0.165,Y -603.071,Z 1389.309,A 0.000,B 0.000,C 90.000,E1 91.547} C_DIS
LIN {X -0.131,Y -597.199,Z 1389.306,A 0.000,B 0.000,C 90.000,E1 91.088} C_DIS
LIN {X -0.177,Y -590.715,Z 1389.304,A 0.000,B 0.000,C 90.000,E1 90.688} C_DIS
LIN {X -0.037,Y -585.411,Z 1389.302,A 0.000,B 0.000,C 90.000,E1 90.401} C_DIS
LIN {X -0.277,Y -577.995,Z 1389.300,A 0.000,B 0.000,C 90.000,E1 90.057} C_DIS
LIN {X -0.113,Y -577.349,Z 1389.300,A 0.000,B 0.000,C 90.000,E1 90.000} C_DIS
LIN {X 0.279,Y -574.336,Z 1389.298,A 0.000,B 0.000,C 90.000,E1 89.656} C_DIS
LIN {X 0.238,Y -574.303,Z 1389.298,A 0.000,B 0.000,C 90.000,E1 89.656} C_DIS
LIN {X 0.008,Y -573.679,Z 1389.297,A 0.000,B 0.000,C 90.000,E1 89.427} C_DIS
LIN {X -0.098,Y -573.665,Z 1389.295,A 0.000,B 0.000,C 90.000,E1 89.026} C_DIS
LIN {X -0.220,Y -575.204,Z 1389.284,A 0.000,B 0.000,C 90.000,E1 87.135} C_DIS
LIN {X -0.177,Y -578.062,Z 1389.267,A 0.000,B 0.000,C 90.000,E1 84.147} C_DIS
LIN {X -0.057,Y -580.243,Z 1389.257,A 0.000,B 0.000,C 90.000,E1 82.243} C_DIS
LIN {X -0.034,Y -582.170,Z 1389.248,A 0.000,B 0.000,C 90.000,E1 80.622} C_DIS
LIN {X -0.116,Y -583.737,Z 1389.240,A 0.000,B 0.000,C 90.000,E1 79.285} C_DIS
LIN {X 0.270,Y -584.824,Z 1389.234,A 0.000,B 0.000,C 90.000,E1 78.173} C_DIS
LIN {X 0.023,Y -586.236,Z 1389.226,A 0.000,B 0.000,C 90.000,E1 76.589} C_DIS
LIN {X 0.013,Y -587.119,Z 1389.220,A 0.000,B 0.000,C 90.000,E1 75.519} C_DIS
LIN {X 0.271,Y -588.039,Z 1389.212,A 0.000,B 0.000,C 90.000,E1 74.157} C_DIS
LIN {X -0.177,Y -588.918,Z 1389.203,A 0.000,B 0.000,C 90.000,E1 72.598} C_DIS
LIN {X -0.184,Y -590.005,Z 1389.193,A 0.000,B 0.000,C 90.000,E1 70.732} C_DIS
LIN {X 0.029,Y -590.597,Z 1389.187,A 0.000,B 0.000,C 90.000,E1 69.645} C_DIS
LIN {X -0.100,Y -591.689,Z 1389.177,A 0.000,B 0.000,C 90.000,E1 67.794} C_DIS
LIN {X 0.030,Y -593.013,Z 1389.166,A 0.000,B 0.000,C 90.000,E1 65.921} C_DIS
LIN {X -0.003,Y -594.282,Z 1389.157,A 0.000,B 0.000,C 90.000,E1 64.332} C_DIS
LIN {X -0.009,Y -595.621,Z 1389.149,A 0.000,B 0.000,C 90.000,E1 62.743} C_DIS
LIN {X 0.219,Y -597.840,Z 1389.134,A 0.000,B 0.000,C 90.000,E1 60.078} C_DIS
LIN {X 0.027,Y -599.569,Z 1389.124,A 0.000,B 0.000,C 90.000,E1 58.250} C_DIS
LIN {X -0.355,Y -600.997,Z 1389.115,A 0.000,B 0.000,C 90.000,E1 56.707} C_DIS
LIN {X -0.301,Y -602.183,Z 1389.108,A 0.000,B 0.000,C 90.000,E1 55.388} C_DIS
LIN {X -0.229,Y -603.400,Z 1389.100,A 0.000,B 0.000,C 90.000,E1 54.069} C_DIS
LIN {X -0.008,Y -604.763,Z 1389.092,A 0.000,B 0.000,C 90.000,E1 52.477} C_DIS
LIN {X -0.020,Y -605.696,Z 1389.084,A 0.000,B 0.000,C 90.000,E1 51.170} C_DIS
LIN {X 0.100,Y -606.288,Z 1389.078,A 0.000,B 0.000,C 90.000,E1 50.114} C_DIS
LIN {X -0.164,Y -606.803,Z 1389.073,A 0.000,B 0.000,C 90.000,E1 49.094} C_DIS
LIN {X -0.294,Y -607.031,Z 1389.068,A 0.000,B 0.000,C 90.000,E1 48.324} C_DIS
LIN {X -0.131,Y -607.333,Z 1389.060,A 0.000,B 0.000,C 90.000,E1 46.743} C_DIS
LIN {X -0.008,Y -607.319,Z 1389.054,A 0.000,B 0.000,C 90.000,E1 45.688} C_DIS
LIN {X -0.333,Y -607.213,Z 1389.048,A 0.000,B 0.000,C 90.000,E1 44.676} C_DIS
LIN {X -0.228,Y -606.882,Z 1389.042,A 0.000,B 0.000,C 90.000,E1 43.623} C_DIS
LIN {X 0.311,Y -606.452,Z 1389.036,A 0.000,B 0.000,C 90.000,E1 42.528} C_DIS
LIN {X 0.042,Y -605.555,Z 1389.028,A 0.000,B 0.000,C 90.000,E1 40.987} C_DIS
LIN {X 0.156,Y -604.828,Z 1389.022,A 0.000,B 0.000,C 90.000,E1 39.930} C_DIS
LIN {X -0.126,Y -603.989,Z 1389.016,A 0.000,B 0.000,C 90.000,E1 38.910} C_DIS
LIN {X -0.156,Y -602.662,Z 1389.009,A 0.000,B 0.000,C 90.000,E1 37.604} C_DIS
LIN {X 0.020,Y -601.253,Z 1389.003,A 0.000,B 0.000,C 90.000,E1 36.537} C_DIS
LIN {X -0.311,Y -599.615,Z 1388.997,A 0.000,B 0.000,C 90.000,E1 35.518} C_DIS
LIN {X 0.069,Y -598.112,Z 1388.993,A 0.000,B 0.000,C 90.000,E1 34.692} C_DIS
LIN {X 0.167,Y -595.792,Z 1388.987,A 0.000,B 0.000,C 90.000,E1 33.627} C_DIS
LIN {X 0.179,Y -593.891,Z 1388.983,A 0.000,B 0.000,C 90.000,E1 32.832} C_DIS
LIN {X -0.115,Y -591.058,Z 1388.977,A 0.000,B 0.000,C 90.000,E1 31.799} C_DIS
LIN {X -0.028,Y -589.418,Z 1388.974,A 0.000,B 0.000,C 90.000,E1 31.258} C_DIS
LIN {X -0.071,Y -586.592,Z 1388.969,A 0.000,B 0.000,C 90.000,E1 30.463} C_DIS
LIN {X -0.018,Y -584.540,Z 1388.966,A 0.000,B 0.000,C 90.000,E1 29.922} C_DIS
LIN {X -0.269,Y -582.304,Z 1388.963,A 0.000,B 0.000,C 90.000,E1 29.411} C_DIS
LIN {X 0.055,Y -577.973,Z 1388.958,A 0.000,B 0.000,C 90.000,E1 28.437} C_DIS
LIN {X 0.036,Y -575.283,Z 1388.955,A 0.000,B 0.000,C 90.000,E1 27.897} C_DIS
LIN {X -0.271,Y -572.388,Z 1388.952,A 0.000,B 0.000,C 90.000,E1 27.385} C_DIS
LIN {X 0.000,Y -567.763,Z 1388.948,A 0.000,B 0.000,C 90.000,E1 26.539} C_DIS
LIN {X 0.060,Y -563.699,Z 1388.944,A 0.000,B 0.000,C 90.000,E1 25.848} C_DIS
LIN {X 0.186,Y -560.240,Z 1388.941,A 0.000,B 0.000,C 90.000,E1 25.283} C_DIS
LIN {X -0.218,Y -556.579,Z 1388.938,A 0.000,B 0.000,C 90.000,E1 24.771} C_DIS
LIN {X -0.140,Y -552.658,Z 1388.934,A 0.000,B 0.000,C 90.000,E1 24.207} C_DIS
LIN {X 0.025,Y -549.591,Z 1388.932,A 0.000,B 0.000,C 90.000,E1 23.770} C_DIS
LIN {X -0.135,Y -541.907,Z 1388.927,A 0.000,B 0.000,C 90.000,E1 22.823} C_DIS
LIN {X 0.191,Y -535.944,Z 1388.923,A 0.000,B 0.000,C 90.000,E1 22.078} C_DIS
LIN {X -0.101,Y -525.734,Z 1388.917,A 0.000,B 0.000,C 90.000,E1 20.972} C_DIS
LIN {X 0.150,Y -520.447,Z 1388.913,A 0.000,B 0.000,C 90.000,E1 20.375} C_DIS
LIN {X -0.178,Y -512.630,Z 1388.909,A 0.000,B 0.000,C 90.000,E1 19.577} C_DIS
LIN {X 0.233,Y -501.731,Z 1388.902,A 0.000,B 0.000,C 90.000,E1 18.417} C_DIS
LIN {X 0.096,Y -485.679,Z 1388.893,A 0.000,B 0.000,C 90.000,E1 16.804} C_DIS
LIN {X -0.257,Y -469.071,Z 1388.884,A 0.000,B 0.000,C 90.000,E1 15.134} C_DIS
LIN {X -0.113,Y -460.631,Z 1388.879,A 0.000,B 0.000,C 90.000,E1 14.245} C_DIS
LIN {X -0.169,Y -448.185,Z 1388.872,A 0.000,B 0.000,C 90.000,E1 12.939} C_DIS
LIN {X -0.067,Y -428.748,Z 1388.860,A 0.000,B 0.000,C 90.000,E1 10.782} C_DIS
LIN {X 0.060,Y -412.336,Z 1388.849,A 0.000,B 0.000,C 90.000,E1 8.803} C_DIS
LIN {X 0.101,Y -399.988,Z 1388.841,A 0.000,B 0.000,C 90.000,E1 7.296} C_DIS
LIN {X 0.145,Y -393.201,Z 1388.836,A 0.000,B 0.000,C 90.000,E1 6.429} C_DIS
LIN {X 0.071,Y -390.996,Z 1388.834,A 0.000,B 0.000,C 90.000,E1 6.087} C_DIS
LIN {X 0.142,Y -390.045,Z 1388.833,A 0.000,B 0.000,C 90.000,E1 5.910} C_DIS
LIN {X 0.104,Y -390.019,Z 1388.833,A 0.000,B 0.000,C 90.000,E1 5.910} C_DIS
LIN {X 0.152,Y -389.954,Z 1388.833,A 0.000,B 0.000,C 90.000,E1 5.853} C_DIS
LIN {X 0.115,Y -389.982,Z 1388.833,A 0.000,B 0.000,C 90.000,E1 5.853} C_DIS
LIN {X -0.026,Y -392.093,Z 1388.831,A 0.000,B 0.000,C 90.000,E1 5.568} C_DIS
LIN {X -0.037,Y -393.632,Z 1388.830,A 0.000,B 0.000,C 90.000,E1 5.391} C_DIS
LIN {X 0.080,Y -405.433,Z 1388.824,A 0.000,B 0.000,C 90.000,E1 4.359} C_DIS
LIN {X 0.188,Y -411.425,Z 1388.821,A 0.000,B 0.000,C 90.000,E1 3.784} C_DIS
LIN {X -0.035,Y -418.211,Z 1388.817,A 0.000,B 0.000,C 90.000,E1 3.037} C_DIS
LIN {X -0.005,Y -424.242,Z 1388.813,A 0.000,B 0.000,C 90.000,E1 2.236} C_DIS
LIN {X 0.156,Y -428.867,Z 1388.809,A 0.000,B 0.000,C 90.000,E1 1.547} C_DIS
LIN {X -0.095,Y -434.471,Z 1388.804,A 0.000,B 0.000,C 90.000,E1 0.745} C_DIS
LIN {X 0.167,Y -440.466,Z 1388.799,A 0.000,B 0.000,C 90.000,E1 359.771} C_DIS
LIN {X -0.039,Y -444.537,Z 1388.795,A 0.000,B 0.000,C 90.000,E1 359.141} C_DIS
LIN {X -0.217,Y -448.419,Z 1388.792,A 0.000,B 0.000,C 90.000,E1 358.511} C_DIS
LIN {X -0.193,Y -453.652,Z 1388.786,A 0.000,B 0.000,C 90.000,E1 357.535} C_DIS
LIN {X -0.192,Y -457.755,Z 1388.782,A 0.000,B 0.000,C 90.000,E1 356.731} C_DIS
LIN {X 0.182,Y -460.821,Z 1388.778,A 0.000,B 0.000,C 90.000,E1 356.045} C_DIS
LIN {X -0.069,Y -464.979,Z 1388.773,A 0.000,B 0.000,C 90.000,E1 355.122} C_DIS
LIN {X -0.205,Y -469.456,Z 1388.767,A 0.000,B 0.000,C 90.000,E1 354.033} C_DIS
LIN {X 0.068,Y -470.614,Z 1388.765,A 0.000,B 0.000,C 90.000,E1 353.685} C_DIS
LIN {X -0.122,Y -471.611,Z 1388.763,A 0.000,B 0.000,C 90.000,E1 353.394} C_DIS
LIN {X 0.106,Y -472.464,Z 1388.761,A 0.000,B 0.000,C 90.000,E1 353.053} C_DIS
LIN {X -0.075,Y -473.054,Z 1388.760,A 0.000,B 0.000,C 90.000,E1 352.761} C_DIS
LIN {X 0.218,Y -473.333,Z 1388.758,A 0.000,B 0.000,C 90.000,E1 352.413} C_DIS
LIN {X -0.019,Y -473.013,Z 1388.756,A 0.000,B 0.000,C 90.000,E1 352.129} C_DIS
LIN {X 0.162,Y -472.275,Z 1388.755,A 0.000,B 0.000,C 90.000,E1 351.951} C_DIS
LIN {X -0.014,Y -471.306,Z 1388.755,A 0.000,B 0.000,C 90.000,E1 351.894} C_DIS
LIN {X 0.114,Y -456.133,Z 1388.753,A 0.000,B 0.000,C 90.000,E1 351.602} C_DIS
LIN {X 0.153,Y -415.789,Z 1388.749,A 0.000,B 0.000,C 90.000,E1 350.792} C_DIS
LIN {X 0.157,Y -379.662,Z 1388.744,A 0.000,B 0.000,C 90.000,E1 349.926} C_DIS
LIN {X -0.151,Y -358.859,Z 1388.741,A 0.000,B 0.000,C 90.000,E1 349.398} C_DIS
LIN {X -0.171,Y -358.753,Z 1388.741,A 0.000,B 0.000,C 90.000,E1 349.398} C_DIS
LIN {X 0.137,Y -359.526,Z 1388.726,A 0.000,B 0.000,C 90.000,E1 346.700} C_DIS
LIN {X -0.135,Y -359.549,Z 1388.716,A 0.000,B 0.000,C 90.000,E1 344.866} C_DIS
LIN {X -0.037,Y -361.973,Z 1388.682,A 0.000,B 0.000,C 90.000,E1 338.847} C_DIS
LIN {X -0.120,Y -365.902,Z 1388.643,A 0.000,B 0.000,C 90.000,E1 331.769} C_DIS
LIN {X -0.040,Y -366.209,Z 1388.641,A 0.000,B 0.000,C 90.000,E1 331.385} C_DIS
LIN {X 0.180,Y -371.263,Z 1388.604,A 0.000,B 0.000,C 90.000,E1 324.689} C_DIS
LIN {X -0.049,Y -371.696,Z 1388.602,A 0.000,B 0.000,C 90.000,E1 324.356} C_DIS
LIN {X -0.004,Y -377.258,Z 1388.567,A 0.000,B 0.000,C 90.000,E1 318.119} C_DIS
LIN {X -0.006,Y -378.183,Z 1388.563,A 0.000,B 0.000,C 90.000,E1 317.391} C_DIS
LIN {X -0.020,Y -383.836,Z 1388.531,A 0.000,B 0.000,C 90.000,E1 311.595} C_DIS
LIN {X 0.064,Y -384.823,Z 1388.527,A 0.000,B 0.000,C 90.000,E1 310.862} C_DIS
LIN {X 0.084,Y -390.997,Z 1388.493,A 0.000,B 0.000,C 90.000,E1 304.771} C_DIS
LIN {X 0.152,Y -391.384,Z 1388.491,A 0.000,B 0.000,C 90.000,E1 304.405} C_DIS
LIN {X 0.096,Y -396.726,Z 1388.460,A 0.000,B 0.000,C 90.000,E1 298.743} C_DIS
LIN {X -0.034,Y -397.087,Z 1388.458,A 0.000,B 0.000,C 90.000,E1 298.409} C_DIS
LIN {X 0.102,Y -401.521,Z 1388.427,A 0.000,B 0.000,C 90.000,E1 292.770} C_DIS
LIN {X 0.135,Y -401.877,Z 1388.421,A 0.000,B 0.000,C 90.000,E1 291.716} C_DIS
LIN {X -0.143,Y -404.592,Z 1388.396,A 0.000,B 0.000,C 90.000,E1 287.221} C_DIS
LIN {X -0.042,Y -404.758,Z 1388.394,A 0.000,B 0.000,C 90.000,E1 286.858} C_DIS
LIN {X -0.135,Y -406.056,Z 1388.365,A 0.000,B 0.000,C 90.000,E1 281.658} C_DIS
LIN {X -0.045,Y -406.125,Z 1388.363,A 0.000,B 0.000,C 90.000,E1 281.299} C_DIS
LIN {X -0.015,Y -405.663,Z 1388.334,A 0.000,B 0.000,C 90.000,E1 276.087} C_DIS
LIN {X -0.010,Y -405.580,Z 1388.332,A 0.000,B 0.000,C 90.000,E1 275.739} C_DIS
LIN {X 0.064,Y -403.539,Z 1388.305,A 0.000,B 0.000,C 90.000,E1 270.859} C_DIS
LIN {X -0.001,Y -403.007,Z 1388.301,A 0.000,B 0.000,C 90.000,E1 270.172} C_DIS
LIN {X -0.179,Y -398.994,Z 1388.272,A 0.000,B 0.000,C 90.000,E1 264.951} C_DIS
LIN {X -0.017,Y -392.901,Z 1388.240,A 0.000,B 0.000,C 90.000,E1 259.285} C_DIS
LIN {X -0.070,Y -391.252,Z 1388.235,A 0.000,B 0.000,C 90.000,E1 258.229} C_DIS
LIN {X 0.124,Y -385.343,Z 1388.209,A 0.000,B 0.000,C 90.000,E1 253.559} C_DIS
LIN {X 0.146,Y -384.911,Z 1388.207,A 0.000,B 0.000,C 90.000,E1 253.196} C_DIS
LIN {X -0.106,Y -378.073,Z 1388.183,A 0.000,B 0.000,C 90.000,E1 248.901} C_DIS
LIN {X 0.123,Y -376.320,Z 1388.175,A 0.000,B 0.000,C 90.000,E1 247.411} C_DIS
LIN {X 0.102,Y -375.792,Z 1388.173,A 0.000,B 0.000,C 90.000,E1 247.050} C_DIS
LIN {X 0.204,Y -369.038,Z 1388.150,A 0.000,B 0.000,C 90.000,E1 242.999} C_DIS
LIN {X 0.107,Y -366.187,Z 1388.138,A 0.000,B 0.000,C 90.000,E1 240.795} C_DIS
LIN {X -0.051,Y -358.786,Z 1388.113,A 0.000,B 0.000,C 90.000,E1 236.342} C_DIS
LIN {X 0.029,Y -355.976,Z 1388.100,A 0.000,B 0.000,C 90.000,E1 234.069} C_DIS
LIN {X -0.165,Y -348.898,Z 1388.075,A 0.000,B 0.000,C 90.000,E1 229.542} C_DIS
LIN {X 0.036,Y -345.819,Z 1388.060,A 0.000,B 0.000,C 90.000,E1 226.824} C_DIS
LIN {X -0.231,Y -339.071,Z 1388.032,A 0.000,B 0.000,C 90.000,E1 221.838} C_DIS
LIN {X -0.147,Y -336.917,Z 1388.019,A 0.000,B 0.000,C 90.000,E1 219.483} C_DIS
LIN {X 0.127,Y -331.251,Z 1387.991,A 0.000,B 0.000,C 90.000,E1 214.326} C_DIS
LIN {X -0.094,Y -329.342,Z 1387.975,A 0.000,B 0.000,C 90.000,E1 211.592} C_DIS
LIN {X 0.006,Y -328.196,Z 1387.969,A 0.000,B 0.000,C 90.000,E1 210.384} C_DIS
LIN {X 0.034,Y -323.959,Z 1387.931,A 0.000,B 0.000,C 90.000,E1 203.590} C_DIS
LIN {X -0.062,Y -323.858,Z 1387.929,A 0.000,B 0.000,C 90.000,E1 203.206} C_DIS
LIN {X -0.154,Y -321.114,Z 1387.882,A 0.000,B 0.000,C 90.000,E1 194.773} C_DIS
LIN {X -0.077,Y -321.105,Z 1387.880,A 0.000,B 0.000,C 90.000,E1 194.356} C_DIS
LIN {X 0.173,Y -320.559,Z 1387.869,A 0.000,B 0.000,C 90.000,E1 192.355} C_DIS
LIN {X 0.155,Y -320.563,Z 1387.869,A 0.000,B 0.000,C 90.000,E1 192.355} C_DIS
LIN {X 0.027,Y -347.841,Z 1387.864,A 0.000,B 0.000,C 90.000,E1 191.422} C_DIS
LIN {X -0.007,Y -377.445,Z 1387.859,A 0.000,B 0.000,C 90.000,E1 190.546} C_DIS
LIN {X 0.206,Y -410.946,Z 1387.854,A 0.000,B 0.000,C 90.000,E1 189.670} C_DIS
LIN {X 0.129,Y -429.683,Z 1387.852,A 0.000,B 0.000,C 90.000,E1 189.265} C_DIS
LIN {X -0.042,Y -432.152,Z 1387.851,A 0.000,B 0.000,C 90.000,E1 189.208} C_DIS
LIN {X -0.056,Y -433.118,Z 1387.851,A 0.000,B 0.000,C 90.000,E1 189.095} C_DIS
LIN {X 0.109,Y -434.266,Z 1387.849,A 0.000,B 0.000,C 90.000,E1 188.746} C_DIS
LIN {X -0.196,Y -434.660,Z 1387.847,A 0.000,B 0.000,C 90.000,E1 188.454} C_DIS
LIN {X -0.068,Y -434.708,Z 1387.845,A 0.000,B 0.000,C 90.000,E1 188.106} C_DIS
LIN {X -0.042,Y -434.328,Z 1387.838,A 0.000,B 0.000,C 90.000,E1 186.777} C_DIS
LIN {X -0.148,Y -433.888,Z 1387.832,A 0.000,B 0.000,C 90.000,E1 185.796} C_DIS
LIN {X 0.052,Y -433.474,Z 1387.828,A 0.000,B 0.000,C 90.000,E1 185.106} C_DIS
LIN {X -0.101,Y -432.533,Z 1387.823,A 0.000,B 0.000,C 90.000,E1 184.131} C_DIS
LIN {X 0.089,Y -431.753,Z 1387.819,A 0.000,B 0.000,C 90.000,E1 183.440} C_DIS
LIN {X -0.007,Y -429.832,Z 1387.812,A 0.000,B 0.000,C 90.000,E1 182.121} C_DIS
LIN {X -0.136,Y -427.265,Z 1387.804,A 0.000,B 0.000,C 90.000,E1 180.802} C_DIS
LIN {X -0.071,Y -426.600,Z 1387.802,A 0.000,B 0.000,C 90.000,E1 180.458} C_DIS
LIN {X 0.110,Y -423.943,Z 1387.797,A 0.000,B 0.000,C 90.000,E1 179.427} C_DIS
LIN {X -0.211,Y -421.971,Z 1387.793,A 0.000,B 0.000,C 90.000,E1 178.797} C_DIS
LIN {X -0.075,Y -418.429,Z 1387.788,A 0.000,B 0.000,C 90.000,E1 177.764} C_DIS
LIN {X -0.017,Y -415.080,Z 1387.783,A 0.000,B 0.000,C 90.000,E1 176.906} C_DIS
LIN {X 0.050,Y -409.971,Z 1387.777,A 0.000,B 0.000,C 90.000,E1 175.869} C_DIS
LIN {X 0.044,Y -405.086,Z 1387.772,A 0.000,B 0.000,C 90.000,E1 175.008} C_DIS
LIN {X -0.002,Y -398.391,Z 1387.767,A 0.000,B 0.000,C 90.000,E1 173.970} C_DIS
LIN {X -0.091,Y -393.756,Z 1387.763,A 0.000,B 0.000,C 90.000,E1 173.280} C_DIS
LIN {X 0.045,Y -384.131,Z 1387.754,A 0.000,B 0.000,C 90.000,E1 171.659} C_DIS
LIN {X -0.013,Y -374.326,Z 1387.744,A 0.000,B 0.000,C 90.000,E1 169.859} C_DIS
LIN {X 0.101,Y -370.031,Z 1387.739,A 0.000,B 0.000,C 90.000,E1 168.926} C_DIS
LIN {X 0.070,Y -367.483,Z 1387.734,A 0.000,B 0.000,C 90.000,E1 168.049} C_DIS
LIN {X 0.033,Y -367.478,Z 1387.734,A 0.000,B 0.000,C 90.000,E1 168.049} C_DIS
LIN {X 0.092,Y -367.626,Z 1387.732,A 0.000,B 0.000,C 90.000,E1 167.757} C_DIS
LIN {X 0.055,Y -367.638,Z 1387.732,A 0.000,B 0.000,C 90.000,E1 167.757} C_DIS
LIN {X -0.002,Y -369.069,Z 1387.730,A 0.000,B 0.000,C 90.000,E1 167.465} C_DIS
LIN {X -0.032,Y -369.780,Z 1387.729,A 0.000,B 0.000,C 90.000,E1 167.285} C_DIS
LIN {X 0.060,Y -375.166,Z 1387.725,A 0.000,B 0.000,C 90.000,E1 166.533} C_DIS
LIN {X -0.091,Y -380.800,Z 1387.722,A 0.000,B 0.000,C 90.000,E1 165.880} C_DIS
LIN {X -0.068,Y -391.285,Z 1387.715,A 0.000,B 0.000,C 90.000,E1 164.755} C_DIS
LIN {X 0.144,Y -405.159,Z 1387.708,A 0.000,B 0.000,C 90.000,E1 163.378} C_DIS
LIN {X -0.176,Y -419.343,Z 1387.701,A 0.000,B 0.000,C 90.000,E1 162.181} C_DIS
LIN {X 0.082,Y -441.472,Z 1387.691,A 0.000,B 0.000,C 90.000,E1 160.369} C_DIS
LIN {X 0.195,Y -455.421,Z 1387.685,A 0.000,B 0.000,C 90.000,E1 159.263} C_DIS
LIN {X 0.016,Y -464.725,Z 1387.681,A 0.000,B 0.000,C 90.000,E1 158.539} C_DIS
LIN {X -0.221,Y -473.712,Z 1387.677,A 0.000,B 0.000,C 90.000,E1 157.794} C_DIS
LIN {X 0.040,Y -481.053,Z 1387.673,A 0.000,B 0.000,C 90.000,E1 157.102} C_DIS
LIN {X 0.035,Y -490.912,Z 1387.668,A 0.000,B 0.000,C 90.000,E1 156.177} C_DIS
LIN {X -0.147,Y -495.104,Z 1387.666,A 0.000,B 0.000,C 90.000,E1 155.793} C_DIS
LIN {X -0.247,Y -501.930,Z 1387.662,A 0.000,B 0.000,C 90.000,E1 155.101} C_DIS
LIN {X -0.132,Y -505.875,Z 1387.659,A 0.000,B 0.000,C 90.000,E1 154.665} C_DIS
LIN {X 0.003,Y -513.537,Z 1387.654,A 0.000,B 0.000,C 90.000,E1 153.768} C_DIS
LIN {X 0.002,Y -519.392,Z 1387.650,A 0.000,B 0.000,C 90.000,E1 153.050} C_DIS
LIN {X -0.195,Y -523.868,Z 1387.647,A 0.000,B 0.000,C 90.000,E1 152.487} C_DIS
LIN {X 0.035,Y -526.953,Z 1387.645,A 0.000,B 0.000,C 90.000,E1 152.025} C_DIS
LIN {X 0.137,Y -530.660,Z 1387.641,A 0.000,B 0.000,C 90.000,E1 151.435} C_DIS
LIN {X 0.008,Y -533.967,Z 1387.638,A 0.000,B 0.000,C 90.000,E1 150.873} C_DIS
LIN {X 0.285,Y -537.484,Z 1387.634,A 0.000,B 0.000,C 90.000,E1 150.127} C_DIS
LIN {X -0.140,Y -540.346,Z 1387.630,A 0.000,B 0.000,C 90.000,E1 149.459} C_DIS
LIN {X 0.055,Y -542.505,Z 1387.627,A 0.000,B 0.000,C 90.000,E1 148.869} C_DIS
LIN {X -0.199,Y -544.397,Z 1387.624,A 0.000,B 0.000,C 90.000,E1 148.329} C_DIS
LIN {X 0.051,Y -546.786,Z 1387.619,A 0.000,B 0.000,C 90.000,E1 147.454} C_DIS
LIN {X -0.133,Y -548.739,Z 1387.615,A 0.000,B 0.000,C 90.000,E1 146.628} C_DIS
LIN {X 0.160,Y -550.409,Z 1387.610,A 0.000,B 0.000,C 90.000,E1 145.754} C_DIS
LIN {X 0.326,Y -551.792,Z 1387.605,A 0.000,B 0.000,C 90.000,E1 144.895} C_DIS
LIN {X 0.191,Y -552.914,Z 1387.601,A 0.000,B 0.000,C 90.000,E1 144.069} C_DIS
LIN {X 0.016,Y -553.966,Z 1387.594,A 0.000,B 0.000,C 90.000,E1 142.970} C_DIS
LIN {X 0.090,Y -555.534,Z 1387.583,A 0.000,B 0.000,C 90.000,E1 141.009} C_DIS
LIN {X -0.041,Y -556.343,Z 1387.577,A 0.000,B 0.000,C 90.000,E1 139.908} C_DIS
LIN {X -0.243,Y -556.830,Z 1387.573,A 0.000,B 0.000,C 90.000,E1 139.094} C_DIS
LIN {X 0.097,Y -557.575,Z 1387.563,A 0.000,B 0.000,C 90.000,E1 137.391} C_DIS
LIN {X 0.048,Y -558.231,Z 1387.554,A 0.000,B 0.000,C 90.000,E1 135.729} C_DIS
LIN {X -0.051,Y -558.762,Z 1387.546,A 0.000,B 0.000,C 90.000,E1 134.352} C_DIS
LIN {X -0.074,Y -559.292,Z 1387.537,A 0.000,B 0.000,C 90.000,E1 132.690} C_DIS
LIN {X -0.048,Y -559.610,Z 1387.528,A 0.000,B 0.000,C 90.000,E1 131.024} C_DIS
LIN {X 0.079,Y -559.978,Z 1387.517,A 0.000,B 0.000,C 90.000,E1 129.072} C_DIS
LIN {X 0.140,Y -561.170,Z 1387.502,A 0.000,B 0.000,C 90.000,E1 126.297} C_DIS
LIN {X -0.005,Y -562.075,Z 1387.499,A 0.000,B 0.000,C 90.000,E1 125.724} C_DIS
LIN {X -0.212,Y -564.301,Z 1387.497,A 0.000,B 0.000,C 90.000,E1 125.391} C_DIS
LIN {X 0.102,Y -565.885,Z 1387.496,A 0.000,B 0.000,C 90.000,E1 125.264} C_DIS
LIN {X 0.011,Y -569.822,Z 1387.495,A 0.000,B 0.000,C 90.000,E1 125.152} C_DIS
LIN {X 0.239,Y -579.226,Z 1387.494,A 0.000,B 0.000,C 90.000,E1 124.898} C_DIS
LIN {X -0.167,Y -585.167,Z 1387.493,A 0.000,B 0.000,C 90.000,E1 124.739} C_DIS
LIN {X -0.017,Y -587.876,Z 1387.492,A 0.000,B 0.000,C 90.000,E1 124.612} C_DIS
LIN {X -0.158,Y -590.627,Z 1387.492,A 0.000,B 0.000,C 90.000,E1 124.485} C_DIS
LIN {X -0.238,Y -593.597,Z 1387.491,A 0.000,B 0.000,C 90.000,E1 124.326} C_DIS
LIN {X 0.171,Y -599.346,Z 1387.489,A 0.000,B 0.000,C 90.000,E1 123.913} C_DIS
LIN {X -0.078,Y -603.629,Z 1387.487,A 0.000,B 0.000,C 90.000,E1 123.627} C_DIS
LIN {X 0.129,Y -609.007,Z 1387.484,A 0.000,B 0.000,C 90.000,E1 123.166} C_DIS
LIN {X -0.016,Y -615.545,Z 1387.481,A 0.000,B 0.000,C 90.000,E1 122.594} C_DIS
LIN {X 0.172,Y -617.990,Z 1387.480,A 0.000,B 0.000,C 90.000,E1 122.339} C_DIS
LIN {X -0.047,Y -623.851,Z 1387.476,A 0.000,B 0.000,C 90.000,E1 121.720} C_DIS
LIN {X -0.054,Y -628.172,Z 1387.473,A 0.000,B 0.000,C 90.000,E1 121.209} C_DIS
LIN {X -0.234,Y -633.165,Z 1387.470,A 0.000,B 0.000,C 90.000,E1 120.590} C_DIS
LIN {X 0.172,Y -637.569,Z 1387.466,A 0.000,B 0.000,C 90.000,E1 119.922} C_DIS
LIN {X -0.261,Y -641.496,Z 1387.463,A 0.000,B 0.000,C 90.000,E1 119.333} C_DIS
LIN {X -0.132,Y -644.057,Z 1387.460,A 0.000,B 0.000,C 90.000,E1 118.821} C_DIS
LIN {X 0.016,Y -646.300,Z 1387.457,A 0.000,B 0.000,C 90.000,E1 118.309} C_DIS
LIN {X 0.096,Y -647.287,Z 1387.456,A 0.000,B 0.000,C 90.000,E1 118.052} C_DIS
LIN {X -0.305,Y -648.764,Z 1387.453,A 0.000,B 0.000,C 90.000,E1 117.590} C_DIS
LIN {X -0.121,Y -649.849,Z 1387.450,A 0.000,B 0.000,C 90.000,E1 117.078} C_DIS
LIN {X -0.026,Y -650.120,Z 1387.449,A 0.000,B 0.000,C 90.000,E1 116.821} C_DIS
LIN {X -0.317,Y -650.214,Z 1387.445,A 0.000,B 0.000,C 90.000,E1 116.104} C_DIS
LIN {X -0.123,Y -649.903,Z 1387.442,A 0.000,B 0.000,C 90.000,E1 115.591} C_DIS
LIN {X 0.067,Y -649.112,Z 1387.439,A 0.000,B 0.000,C 90.000,E1 115.079} C_DIS
LIN {X 0.159,Y -648.584,Z 1387.438,A 0.000,B 0.000,C 90.000,E1 114.823} C_DIS
LIN {X 0.070,Y -646.577,Z 1387.435,A 0.000,B 0.000,C 90.000,E1 114.335} C_DIS
LIN {X 0.112,Y -645.919,Z 1387.435,A 0.000,B 0.000,C 90.000,E1 114.207} C_DIS
LIN {X 0.269,Y -642.224,Z 1387.432,A 0.000,B 0.000,C 90.000,E1 113.695} C_DIS
LIN {X 0.048,Y -640.856,Z 1387.431,A 0.000,B 0.000,C 90.000,E1 113.590} C_DIS
LIN {X 0.275,Y -636.708,Z 1387.430,A 0.000,B 0.000,C 90.000,E1 113.334} C_DIS
LIN {X -0.195,Y -633.989,Z 1387.429,A 0.000,B 0.000,C 90.000,E1 113.206} C_DIS
LIN {X 0.170,Y -631.773,Z 1387.428,A 0.000,B 0.000,C 90.000,E1 113.078} C_DIS
LIN {X -0.136,Y -621.975,Z 1387.427,A 0.000,B 0.000,C 90.000,E1 112.770} C_DIS
LIN {X 0.190,Y -611.060,Z 1387.425,A 0.000,B 0.000,C 90.000,E1 112.408} C_DIS
LIN {X 0.156,Y -611.048,Z 1387.425,A 0.000,B 0.000,C 90.000,E1 112.408} C_DIS
LIN {X 0.258,Y -614.372,Z 1387.423,A 0.000,B 0.000,C 90.000,E1 112.078} C_DIS
LIN {X -0.206,Y -622.602,Z 1387.419,A 0.000,B 0.000,C 90.000,E1 111.354} C_DIS
LIN {X 0.031,Y -626.255,Z 1387.417,A 0.000,B 0.000,C 90.000,E1 110.972} C_DIS
LIN {X -0.164,Y -629.868,Z 1387.414,A 0.000,B 0.000,C 90.000,E1 110.610} C_DIS
LIN {X 0.263,Y -635.188,Z 1387.411,A 0.000,B 0.000,C 90.000,E1 109.939} C_DIS
LIN {X 0.115,Y -639.888,Z 1387.407,A 0.000,B 0.000,C 90.000,E1 109.322} C_DIS
LIN {X -0.209,Y -644.051,Z 1387.404,A 0.000,B 0.000,C 90.000,E1 108.725} C_DIS
LIN {X 0.146,Y -648.480,Z 1387.400,A 0.000,B 0.000,C 90.000,E1 107.946} C_DIS
LIN {X -0.070,Y -652.279,Z 1387.396,A 0.000,B 0.000,C 90.000,E1 107.221} C_DIS
LIN {X -0.262,Y -655.261,Z 1387.392,A 0.000,B 0.000,C 90.000,E1 106.496} C_DIS
LIN {X 0.133,Y -656.669,Z 1387.389,A 0.000,B 0.000,C 90.000,E1 105.969} C_DIS
LIN {X 0.199,Y -657.284,Z 1387.387,A 0.000,B 0.000,C 90.000,E1 105.717} C_DIS
LIN {X -0.023,Y -658.278,Z 1387.385,A 0.000,B 0.000,C 90.000,E1 105.245} C_DIS
LIN {X 0.197,Y -659.777,Z 1387.379,A 0.000,B 0.000,C 90.000,E1 104.245} C_DIS
LIN {X -0.102,Y -660.569,Z 1387.375,A 0.000,B 0.000,C 90.000,E1 103.536} C_DIS
LIN {X 0.249,Y -660.890,Z 1387.371,A 0.000,B 0.000,C 90.000,E1 102.771} C_DIS
LIN {X 0.055,Y -660.865,Z 1387.368,A 0.000,B 0.000,C 90.000,E1 102.299} C_DIS
LIN {X -0.142,Y -660.657,Z 1387.366,A 0.000,B 0.000,C 90.000,E1 101.827} C_DIS
LIN {X 0.074,Y -659.904,Z 1387.362,A 0.000,B 0.000,C 90.000,E1 101.074} C_DIS
LIN {X -0.132,Y -659.229,Z 1387.359,A 0.000,B 0.000,C 90.000,E1 100.602} C_DIS
LIN {X 0.077,Y -657.656,Z 1387.355,A 0.000,B 0.000,C 90.000,E1 99.849} C_DIS
LIN {X -0.151,Y -656.432,Z 1387.352,A 0.000,B 0.000,C 90.000,E1 99.378} C_DIS
LIN {X 0.152,Y -654.978,Z 1387.349,A 0.000,B 0.000,C 90.000,E1 98.859} C_DIS
LIN {X -0.196,Y -653.310,Z 1387.347,A 0.000,B 0.000,C 90.000,E1 98.398} C_DIS
LIN {X 0.184,Y -651.458,Z 1387.344,A 0.000,B 0.000,C 90.000,E1 97.871} C_DIS
LIN {X 0.227,Y -648.170,Z 1387.340,A 0.000,B 0.000,C 90.000,E1 97.125} C_DIS
LIN {X -0.043,Y -646.396,Z 1387.338,A 0.000,B 0.000,C 90.000,E1 96.777} C_DIS
LIN {X -0.098,Y -641.673,Z 1387.333,A 0.000,B 0.000,C 90.000,E1 95.910} C_DIS
LIN {X -0.275,Y -636.497,Z 1387.328,A 0.000,B 0.000,C 90.000,E1 95.049} C_DIS
LIN {X -0.105,Y -633.287,Z 1387.325,A 0.000,B 0.000,C 90.000,E1 94.531} C_DIS
LIN {X 0.038,Y -629.749,Z 1387.322,A 0.000,B 0.000,C 90.000,E1 94.012} C_DIS
LIN {X 0.113,Y -625.595,Z 1387.320,A 0.000,B 0.000,C 90.000,E1 93.498} C_DIS
LIN {X 0.218,Y -620.737,Z 1387.317,A 0.000,B 0.000,C 90.000,E1 92.980} C_DIS
LIN {X -0.266,Y -614.154,Z 1387.313,A 0.000,B 0.000,C 90.000,E1 92.407} C_DIS
LIN {X 0.234,Y -607.591,Z 1387.310,A 0.000,B 0.000,C 90.000,E1 91.776} C_DIS
LIN {X 0.134,Y -603.508,Z 1387.308,A 0.000,B 0.000,C 90.000,E1 91.432} C_DIS
LIN {X 0.091,Y -599.012,Z 1387.306,A 0.000,B 0.000,C 90.000,E1 91.088} C_DIS
LIN {X 0.226,Y -595.906,Z 1387.305,A 0.000,B 0.000,C 90.000,E1 90.859} C_DIS
LIN {X 0.139,Y -590.996,Z 1387.303,A 0.000,B 0.000,C 90.000,E1 90.573} C_DIS
LIN {X 0.031,Y -587.552,Z 1387.302,A 0.000,B 0.000,C 90.000,E1 90.401} C_DIS
LIN {X 0.251,Y -578.490,Z 1387.300,A 0.000,B 0.000,C 90.000,E1 89.943} C_DIS
LIN {X -0.164,Y -577.778,Z 1387.300,A 0.000,B 0.000,C 90.000,E1 89.943} C_DIS
LIN {X -0.032,Y -574.425,Z 1387.298,A 0.000,B 0.000,C 90.000,E1 89.599} C_DIS
LIN {X -0.073,Y -574.408,Z 1387.298,A 0.000,B 0.000,C 90.000,E1 89.599} C_DIS
LIN {X -0.001,Y -573.795,Z 1387.297,A 0.000,B 0.000,C 90.000,E1 89.370} C_DIS
LIN {X 0.145,Y -573.689,Z 1387.295,A 0.000,B 0.000,C 90.000,E1 89.083} C_DIS
LIN {X -0.143,Y -573.949,Z 1387.292,A 0.000,B 0.000,C 90.000,E1 88.568} C_DIS
LIN {X 0.022,Y -575.079,Z 1387.284,A 0.000,B 0.000,C 90.000,E1 87.192} C_DIS
LIN {X -0.279,Y -577.312,Z 1387.271,A 0.000,B 0.000,C 90.000,E1 84.780} C_DIS
LIN {X -0.032,Y -579.761,Z 1387.259,A 0.000,B 0.000,C 90.000,E1 82.591} C_DIS
LIN {X -0.020,Y -581.702,Z 1387.250,A 0.000,B 0.000,C 90.000,E1 80.971} C_DIS
LIN {X 0.126,Y -583.614,Z 1387.241,A 0.000,B 0.000,C 90.000,E1 79.342} C_DIS
LIN {X -0.060,Y -584.684,Z 1387.235,A 0.000,B 0.000,C 90.000,E1 78.285} C_DIS
LIN {X 0.020,Y -585.922,Z 1387.228,A 0.000,B 0.000,C 90.000,E1 76.937} C_DIS
LIN {X 0.113,Y -587.034,Z 1387.220,A 0.000,B 0.000,C 90.000,E1 75.589} C_DIS
LIN {X 0.199,Y -588.094,Z 1387.211,A 0.000,B 0.000,C 90.000,E1 73.976} C_DIS
LIN {X -0.246,Y -588.992,Z 1387.202,A 0.000,B 0.000,C 90.000,E1 72.417} C_DIS
LIN {X -0.251,Y -590.076,Z 1387.192,A 0.000,B 0.000,C 90.000,E1 70.550} C_DIS
LIN {X -0.157,Y -590.789,Z 1387.184,A 0.000,B 0.000,C 90.000,E1 69.209} C_DIS
LIN {X 0.272,Y -591.458,Z 1387.179,A 0.000,B 0.000,C 90.000,E1 68.103} C_DIS
LIN {X -0.144,Y -592.723,Z 1387.168,A 0.000,B 0.000,C 90.000,E1 66.282} C_DIS
LIN {X 0.110,Y -594.030,Z 1387.159,A 0.000,B 0.000,C 90.000,E1 64.665} C_DIS
LIN {X 0.001,Y -595.544,Z 1387.149,A 0.000,B 0.000,C 90.000,E1 62.820} C_DIS
LIN {X -0.176,Y -598.242,Z 1387.131,A 0.000,B 0.000,C 90.000,E1 59.665} C_DIS
LIN {X -0.072,Y -599.738,Z 1387.123,A 0.000,B 0.000,C 90.000,E1 58.074} C_DIS
LIN {X -0.045,Y -600.935,Z 1387.115,A 0.000,B 0.000,C 90.000,E1 56.755} C_DIS
LIN {X 0.173,Y -602.614,Z 1387.105,A 0.000,B 0.000,C 90.000,E1 54.895} C_DIS
LIN {X -0.235,Y -603.793,Z 1387.098,A 0.000,B 0.000,C 90.000,E1 53.623} C_DIS
LIN {X 0.217,Y -604.906,Z 1387.091,A 0.000,B 0.000,C 90.000,E1 52.271} C_DIS
LIN {X 0.204,Y -605.809,Z 1387.083,A 0.000,B 0.000,C 90.000,E1 50.964} C_DIS
LIN {X 0.123,Y -606.518,Z 1387.076,A 0.000,B 0.000,C 90.000,E1 49.666} C_DIS
LIN {X 0.259,Y -606.999,Z 1387.070,A 0.000,B 0.000,C 90.000,E1 48.609} C_DIS
LIN {X -0.175,Y -607.334,Z 1387.060,A 0.000,B 0.000,C 90.000,E1 46.824} C_DIS
LIN {X 0.373,Y -607.344,Z 1387.054,A 0.000,B 0.000,C 90.000,E1 45.729} C_DIS
LIN {X 0.294,Y -607.212,Z 1387.047,A 0.000,B 0.000,C 90.000,E1 44.433} C_DIS
LIN {X -0.208,Y -606.728,Z 1387.040,A 0.000,B 0.000,C 90.000,E1 43.176} C_DIS
LIN {X 0.268,Y -606.554,Z 1387.037,A 0.000,B 0.000,C 90.000,E1 42.609} C_DIS
LIN {X -0.197,Y -605.488,Z 1387.027,A 0.000,B 0.000,C 90.000,E1 40.825} C_DIS
LIN {X 0.171,Y -604.538,Z 1387.020,A 0.000,B 0.000,C 90.000,E1 39.483} C_DIS
LIN {X 0.100,Y -603.873,Z 1387.015,A 0.000,B 0.000,C 90.000,E1 38.705} C_DIS
LIN {X 0.183,Y -602.855,Z 1387.009,A 0.000,B 0.000,C 90.000,E1 37.649} C_DIS
LIN {X 0.354,Y -601.479,Z 1387.003,A 0.000,B 0.000,C 90.000,E1 36.583} C_DIS
LIN {X 0.261,Y -600.305,Z 1386.999,A 0.000,B 0.000,C 90.000,E1 35.804} C_DIS
LIN {X 0.157,Y -598.924,Z 1386.995,A 0.000,B 0.000,C 90.000,E1 35.025} C_DIS
LIN {X 0.035,Y -597.318,Z 1386.990,A 0.000,B 0.000,C 90.000,E1 34.246} C_DIS
LIN {X -0.321,Y -594.233,Z 1386.983,A 0.000,B 0.000,C 90.000,E1 32.959} C_DIS
LIN {X -0.108,Y -591.444,Z 1386.977,A 0.000,B 0.000,C 90.000,E1 31.878} C_DIS
LIN {X 0.177,Y -588.993,Z 1386.973,A 0.000,B 0.000,C 90.000,E1 31.052} C_DIS
LIN {X 0.007,Y -585.034,Z 1386.967,A 0.000,B 0.000,C 90.000,E1 30.001} C_DIS
LIN {X -0.081,Y -581.647,Z 1386.962,A 0.000,B 0.000,C 90.000,E1 29.205} C_DIS
LIN {X 0.230,Y -577.298,Z 1386.957,A 0.000,B 0.000,C 90.000,E1 28.231} C_DIS
LIN {X -0.217,Y -573.051,Z 1386.953,A 0.000,B 0.000,C 90.000,E1 27.462} C_DIS
LIN {X 0.064,Y -568.445,Z 1386.948,A 0.000,B 0.000,C 90.000,E1 26.616} C_DIS
LIN {X 0.041,Y -563.566,Z 1386.943,A 0.000,B 0.000,C 90.000,E1 25.796} C_DIS
LIN {X 0.070,Y -559.185,Z 1386.940,A 0.000,B 0.000,C 90.000,E1 25.103} C_DIS
LIN {X 0.291,Y -554.509,Z 1386.936,A 0.000,B 0.000,C 90.000,E1 24.387} C_DIS
LIN {X 0.233,Y -549.409,Z 1386.932,A 0.000,B 0.000,C 90.000,E1 23.695} C_DIS
LIN {X 0.032,Y -540.358,Z 1386.926,A 0.000,B 0.000,C 90.000,E1 22.589} C_DIS
LIN {X 0.128,Y -536.831,Z 1386.923,A 0.000,B 0.000,C 90.000,E1 22.153} C_DIS
LIN {X -0.086,Y -525.502,Z 1386.916,A 0.000,B 0.000,C 90.000,E1 20.918} C_DIS
LIN {X -0.003,Y -521.592,Z 1386.914,A 0.000,B 0.000,C 90.000,E1 20.482} C_DIS
LIN {X 0.041,Y -512.383,Z 1386.908,A 0.000,B 0.000,C 90.000,E1 19.504} C_DIS
LIN {X 0.118,Y -501.853,Z 1386.902,A 0.000,B 0.000,C 90.000,E1 18.417} C_DIS
LIN {X -0.185,Y -485.573,Z 1386.893,A 0.000,B 0.000,C 90.000,E1 16.804} C_DIS
LIN {X 0.007,Y -468.896,Z 1386.884,A 0.000,B 0.000,C 90.000,E1 15.064} C_DIS
LIN {X -0.153,Y -458.986,Z 1386.878,A 0.000,B 0.000,C 90.000,E1 14.064} C_DIS
LIN {X -0.111,Y -447.829,Z 1386.872,A 0.000,B 0.000,C 90.000,E1 12.883} C_DIS
LIN {X 0.205,Y -427.025,Z 1386.859,A 0.000,B 0.000,C 90.000,E1 10.546} C_DIS
LIN {X -0.158,Y -410.570,Z 1386.848,A 0.000,B 0.000,C 90.000,E1 8.624} C_DIS
LIN {X -0.147,Y -392.768,Z 1386.836,A 0.000,B 0.000,C 90.000,E1 6.429} C_DIS
LIN {X -0.082,Y -390.143,Z 1386.833,A 0.000,B 0.000,C 90.000,E1 5.967} C_DIS
LIN {X -0.121,Y -390.116,Z 1386.833,A 0.000,B 0.000,C 90.000,E1 5.967} C_DIS
LIN {X -0.158,Y -390.109,Z 1386.833,A 0.000,B 0.000,C 90.000,E1 5.967} C_DIS
LIN {X 0.192,Y -390.141,Z 1386.833,A 0.000,B 0.000,C 90.000,E1 5.910} C_DIS
LIN {X -0.185,Y -392.104,Z 1386.831,A 0.000,B 0.000,C 90.000,E1 5.682} C_DIS
LIN {X -0.069,Y -393.984,Z 1386.830,A 0.000,B 0.000,C 90.000,E1 5.454} C_DIS
LIN {X 0.145,Y -399.586,Z 1386.828,A 0.000,B 0.000,C 90.000,E1 4.935} C_DIS
LIN {X 0.179,Y -403.845,Z 1386.826,A 0.000,B 0.000,C 90.000,E1 4.588} C_DIS
LIN {X 0.000,Y -409.875,Z 1386.823,A 0.000,B 0.000,C 90.000,E1 4.073} C_DIS
LIN {X -0.175,Y -414.127,Z 1386.820,A 0.000,B 0.000,C 90.000,E1 3.669} C_DIS
LIN {X -0.130,Y -418.064,Z 1386.818,A 0.000,B 0.000,C 90.000,E1 3.212} C_DIS
LIN {X 0.124,Y -423.165,Z 1386.814,A 0.000,B 0.000,C 90.000,E1 2.522} C_DIS
LIN {X -0.170,Y -429.238,Z 1386.809,A 0.000,B 0.000,C 90.000,E1 1.718} C_DIS
LIN {X 0.012,Y -434.952,Z 1386.805,A 0.000,B 0.000,C 90.000,E1 0.859} C_DIS
LIN {X 0.000,Y -440.533,Z 1386.800,A 0.000,B 0.000,C 90.000,E1 360.000} C_DIS
LIN {X -0.028,Y -445.919,Z 1386.795,A 0.000,B 0.000,C 90.000,E1 359.141} C_DIS
LIN {X -0.196,Y -449.804,Z 1386.792,A 0.000,B 0.000,C 90.000,E1 358.511} C_DIS
LIN {X -0.155,Y -455.071,Z 1386.786,A 0.000,B 0.000,C 90.000,E1 357.535} C_DIS
LIN {X -0.139,Y -459.175,Z 1386.782,A 0.000,B 0.000,C 90.000,E1 356.731} C_DIS
LIN {X -0.214,Y -462.240,Z 1386.778,A 0.000,B 0.000,C 90.000,E1 356.102} C_DIS
LIN {X -0.133,Y -465.792,Z 1386.774,A 0.000,B 0.000,C 90.000,E1 355.298} C_DIS
LIN {X 0.139,Y -469.658,Z 1386.769,A 0.000,B 0.000,C 90.000,E1 354.318} C_DIS
LIN {X 0.177,Y -472.110,Z 1386.765,A 0.000,B 0.000,C 90.000,E1 353.685} C_DIS
LIN {X -0.244,Y -474.400,Z 1386.762,A 0.000,B 0.000,C 90.000,E1 353.109} C_DIS
LIN {X 0.051,Y -475.399,Z 1386.760,A 0.000,B 0.000,C 90.000,E1 352.761} C_DIS
LIN {X -0.118,Y -476.248,Z 1386.758,A 0.000,B 0.000,C 90.000,E1 352.470} C_DIS
LIN {X 0.125,Y -476.875,Z 1386.756,A 0.000,B 0.000,C 90.000,E1 352.129} C_DIS
LIN {X -0.037,Y -477.207,Z 1386.755,A 0.000,B 0.000,C 90.000,E1 351.837} C_DIS
LIN {X -0.196,Y -477.102,Z 1386.753,A 0.000,B 0.000,C 90.000,E1 351.546} C_DIS
LIN {X -0.074,Y -476.705,Z 1386.752,A 0.000,B 0.000,C 90.000,E1 351.376} C_DIS
LIN {X 0.119,Y -475.698,Z 1386.751,A 0.000,B 0.000,C 90.000,E1 351.197} C_DIS
LIN {X -0.082,Y -473.281,Z 1386.751,A 0.000,B 0.000,C 90.000,E1 351.141} C_DIS
LIN {X 0.158,Y -432.152,Z 1386.746,A 0.000,B 0.000,C 90.000,E1 350.274} C_DIS
LIN {X 0.180,Y -396.226,Z 1386.741,A 0.000,B 0.000,C 90.000,E1 349.398} C_DIS
LIN {X -0.119,Y -364.182,Z 1386.736,A 0.000,B 0.000,C 90.000,E1 348.522} C_DIS
LIN {X -0.027,Y -358.964,Z 1386.735,A 0.000,B 0.000,C 90.000,E1 348.342} C_DIS
LIN {X -0.050,Y -358.962,Z 1386.735,A 0.000,B 0.000,C 90.000,E1 348.342} C_DIS
LIN {X 0.104,Y -359.504,Z 1386.727,A 0.000,B 0.000,C 90.000,E1 346.756} C_DIS
LIN {X 0.187,Y -359.542,Z 1386.722,A 0.000,B 0.000,C 90.000,E1 345.992} C_DIS
LIN {X -0.056,Y -361.962,Z 1386.683,A 0.000,B 0.000,C 90.000,E1 338.901} C_DIS
LIN {X -0.042,Y -366.190,Z 1386.641,A 0.000,B 0.000,C 90.000,E1 331.435} C_DIS
LIN {X -0.017,Y -371.206,Z 1386.604,A 0.000,B 0.000,C 90.000,E1 324.769} C_DIS
LIN {X -0.030,Y -371.638,Z 1386.602,A 0.000,B 0.000,C 90.000,E1 324.402} C_DIS
LIN {X 0.027,Y -376.743,Z 1386.570,A 0.000,B 0.000,C 90.000,E1 318.528} C_DIS
LIN {X -0.217,Y -378.138,Z 1386.564,A 0.000,B 0.000,C 90.000,E1 317.472} C_DIS
LIN {X -0.197,Y -384.259,Z 1386.529,A 0.000,B 0.000,C 90.000,E1 311.310} C_DIS
LIN {X 0.099,Y -384.763,Z 1386.527,A 0.000,B 0.000,C 90.000,E1 310.906} C_DIS
LIN {X 0.089,Y -390.930,Z 1386.494,A 0.000,B 0.000,C 90.000,E1 304.818} C_DIS
LIN {X -0.065,Y -391.356,Z 1386.492,A 0.000,B 0.000,C 90.000,E1 304.485} C_DIS
LIN {X 0.106,Y -397.065,Z 1386.458,A 0.000,B 0.000,C 90.000,E1 298.437} C_DIS
LIN {X 0.061,Y -401.467,Z 1386.427,A 0.000,B 0.000,C 90.000,E1 292.823} C_DIS
LIN {X 0.142,Y -401.679,Z 1386.425,A 0.000,B 0.000,C 90.000,E1 292.461} C_DIS
LIN {X 0.188,Y -404.550,Z 1386.396,A 0.000,B 0.000,C 90.000,E1 287.221} C_DIS
LIN {X -0.098,Y -404.762,Z 1386.394,A 0.000,B 0.000,C 90.000,E1 286.913} C_DIS
LIN {X -0.202,Y -406.029,Z 1386.365,A 0.000,B 0.000,C 90.000,E1 281.715} C_DIS
LIN {X -0.192,Y -406.145,Z 1386.363,A 0.000,B 0.000,C 90.000,E1 281.366} C_DIS
LIN {X -0.087,Y -405.651,Z 1386.334,A 0.000,B 0.000,C 90.000,E1 276.144} C_DIS
LIN {X -0.083,Y -405.613,Z 1386.332,A 0.000,B 0.000,C 90.000,E1 275.796} C_DIS
LIN {X -0.009,Y -403.553,Z 1386.305,A 0.000,B 0.000,C 90.000,E1 270.917} C_DIS
LIN {X -0.074,Y -403.059,Z 1386.301,A 0.000,B 0.000,C 90.000,E1 270.229} C_DIS
LIN {X 0.150,Y -399.018,Z 1386.272,A 0.000,B 0.000,C 90.000,E1 264.951} C_DIS
LIN {X 0.067,Y -398.129,Z 1386.268,A 0.000,B 0.000,C 90.000,E1 264.261} C_DIS
LIN {X -0.076,Y -392.936,Z 1386.241,A 0.000,B 0.000,C 90.000,E1 259.342} C_DIS
LIN {X -0.118,Y -392.484,Z 1386.239,A 0.000,B 0.000,C 90.000,E1 258.993} C_DIS
LIN {X 0.030,Y -386.127,Z 1386.213,A 0.000,B 0.000,C 90.000,E1 254.338} C_DIS
LIN {X -0.009,Y -384.997,Z 1386.207,A 0.000,B 0.000,C 90.000,E1 253.268} C_DIS
LIN {X -0.136,Y -378.137,Z 1386.183,A 0.000,B 0.000,C 90.000,E1 248.954} C_DIS
LIN {X 0.077,Y -375.887,Z 1386.173,A 0.000,B 0.000,C 90.000,E1 247.102} C_DIS
LIN {X 0.028,Y -369.109,Z 1386.151,A 0.000,B 0.000,C 90.000,E1 243.076} C_DIS
LIN {X 0.106,Y -366.261,Z 1386.138,A 0.000,B 0.000,C 90.000,E1 240.845} C_DIS
LIN {X 0.067,Y -358.856,Z 1386.113,A 0.000,B 0.000,C 90.000,E1 236.373} C_DIS
LIN {X 0.056,Y -356.045,Z 1386.101,A 0.000,B 0.000,C 90.000,E1 234.116} C_DIS
LIN {X 0.052,Y -348.482,Z 1386.073,A 0.000,B 0.000,C 90.000,E1 229.175} C_DIS
LIN {X 0.112,Y -345.902,Z 1386.061,A 0.000,B 0.000,C 90.000,E1 226.863} C_DIS
LIN {X 0.079,Y -339.126,Z 1386.033,A 0.000,B 0.000,C 90.000,E1 221.838} C_DIS
LIN {X 0.162,Y -336.959,Z 1386.020,A 0.000,B 0.000,C 90.000,E1 219.483} C_DIS
LIN {X 0.016,Y -334.035,Z 1386.006,A 0.000,B 0.000,C 90.000,E1 217.156} C_DIS
LIN {X 0.040,Y -329.371,Z 1385.976,A 0.000,B 0.000,C 90.000,E1 211.623} C_DIS
LIN {X -0.057,Y -328.650,Z 1385.971,A 0.000,B 0.000,C 90.000,E1 210.846} C_DIS
LIN {X -0.159,Y -324.093,Z 1385.934,A 0.000,B 0.000,C 90.000,E1 204.079} C_DIS
LIN {X -0.055,Y -323.870,Z 1385.929,A 0.000,B 0.000,C 90.000,E1 203.259} C_DIS
LIN {X 0.119,Y -323.118,Z 1385.922,A 0.000,B 0.000,C 90.000,E1 202.025} C_DIS
LIN {X -0.083,Y -321.125,Z 1385.880,A 0.000,B 0.000,C 90.000,E1 194.411} C_DIS
LIN {X -0.012,Y -320.833,Z 1385.875,A 0.000,B 0.000,C 90.000,E1 193.536} C_DIS
LIN {X -0.041,Y -320.934,Z 1385.875,A 0.000,B 0.000,C 90.000,E1 193.536} C_DIS
LIN {X 0.134,Y -347.689,Z 1385.870,A 0.000,B 0.000,C 90.000,E1 192.479} C_DIS
LIN {X 0.027,Y -377.119,Z 1385.864,A 0.000,B 0.000,C 90.000,E1 191.535} C_DIS
LIN {X 0.104,Y -410.352,Z 1385.859,A 0.000,B 0.000,C 90.000,E1 190.602} C_DIS
LIN {X 0.026,Y -432.607,Z 1385.856,A 0.000,B 0.000,C 90.000,E1 190.074} C_DIS
LIN {X -0.188,Y -434.502,Z 1385.856,A 0.000,B 0.000,C 90.000,E1 190.018} C_DIS
LIN {X -0.089,Y -435.553,Z 1385.855,A 0.000,B 0.000,C 90.000,E1 189.849} C_DIS
LIN {X 0.042,Y -436.538,Z 1385.853,A 0.000,B 0.000,C 90.000,E1 189.500} C_DIS
LIN {X 0.177,Y -436.939,Z 1385.851,A 0.000,B 0.000,C 90.000,E1 189.151} C_DIS
LIN {X -0.116,Y -437.054,Z 1385.849,A 0.000,B 0.000,C 90.000,E1 188.859} C_DIS
LIN {X 0.163,Y -436.853,Z 1385.845,A 0.000,B 0.000,C 90.000,E1 188.163} C_DIS
LIN {X 0.221,Y -436.476,Z 1385.838,A 0.000,B 0.000,C 90.000,E1 186.834} C_DIS
LIN {X -0.207,Y -435.898,Z 1385.831,A 0.000,B 0.000,C 90.000,E1 185.568} C_DIS
LIN {X -0.078,Y -435.749,Z 1385.829,A 0.000,B 0.000,C 90.000,E1 185.220} C_DIS
LIN {X -0.206,Y -434.967,Z 1385.823,A 0.000,B 0.000,C 90.000,E1 184.245} C_DIS
LIN {X 0.004,Y -434.321,Z 1385.820,A 0.000,B 0.000,C 90.000,E1 183.555} C_DIS
LIN {X 0.033,Y -432.046,Z 1385.811,A 0.000,B 0.000,C 90.000,E1 181.892} C_DIS
LIN {X -0.139,Y -430.242,Z 1385.805,A 0.000,B 0.000,C 90.000,E1 180.917} C_DIS
LIN {X 0.014,Y -428.866,Z 1385.801,A 0.000,B 0.000,C 90.000,E1 180.229} C_DIS
LIN {X -0.204,Y -426.260,Z 1385.796,A 0.000,B 0.000,C 90.000,E1 179.255} C_DIS
LIN {X -0.084,Y -424.382,Z 1385.792,A 0.000,B 0.000,C 90.000,E1 178.568} C_DIS
LIN {X 0.057,Y -421.434,Z 1385.787,A 0.000,B 0.000,C 90.000,E1 177.707} C_DIS
LIN {X 0.145,Y -418.155,Z 1385.783,A 0.000,B 0.000,C 90.000,E1 176.849} C_DIS
LIN {X -0.165,Y -413.165,Z 1385.777,A 0.000,B 0.000,C 90.000,E1 175.869} C_DIS
LIN {X -0.139,Y -408.397,Z 1385.772,A 0.000,B 0.000,C 90.000,E1 175.008} C_DIS
LIN {X -0.142,Y -401.809,Z 1385.766,A 0.000,B 0.000,C 90.000,E1 173.970} C_DIS
LIN {X 0.095,Y -391.514,Z 1385.758,A 0.000,B 0.000,C 90.000,E1 172.356} C_DIS
LIN {X 0.096,Y -379.199,Z 1385.746,A 0.000,B 0.000,C 90.000,E1 170.208} C_DIS
LIN {X -0.180,Y -374.496,Z 1385.741,A 0.000,B 0.000,C 90.000,E1 169.342} C_DIS
LIN {X 0.031,Y -371.227,Z 1385.737,A 0.000,B 0.000,C 90.000,E1 168.578} C_DIS
LIN {X -0.127,Y -369.663,Z 1385.734,A 0.000,B 0.000,C 90.000,E1 168.105} C_DIS
LIN {X 0.131,Y -369.289,Z 1385.733,A 0.000,B 0.000,C 90.000,E1 167.881} C_DIS
LIN {X 0.168,Y -369.147,Z 1385.732,A 0.000,B 0.000,C 90.000,E1 167.645} C_DIS
LIN {X 0.130,Y -369.153,Z 1385.732,A 0.000,B 0.000,C 90.000,E1 167.645} C_DIS
LIN {X 0.175,Y -370.457,Z 1385.729,A 0.000,B 0.000,C 90.000,E1 167.229} C_DIS
LIN {X -0.195,Y -373.587,Z 1385.727,A 0.000,B 0.000,C 90.000,E1 166.825} C_DIS
LIN {X 0.145,Y -374.783,Z 1385.726,A 0.000,B 0.000,C 90.000,E1 166.589} C_DIS
LIN {X -0.205,Y -380.950,Z 1385.721,A 0.000,B 0.000,C 90.000,E1 165.880} C_DIS
LIN {X -0.042,Y -393.003,Z 1385.714,A 0.000,B 0.000,C 90.000,E1 164.574} C_DIS
LIN {X -0.014,Y -405.348,Z 1385.708,A 0.000,B 0.000,C 90.000,E1 163.378} C_DIS
LIN {X 0.124,Y -417.899,Z 1385.702,A 0.000,B 0.000,C 90.000,E1 162.253} C_DIS
LIN {X -0.101,Y -440.069,Z 1385.692,A 0.000,B 0.000,C 90.000,E1 160.496} C_DIS
LIN {X 0.022,Y -454.018,Z 1385.686,A 0.000,B 0.000,C 90.000,E1 159.390} C_DIS
LIN {X 0.045,Y -461.742,Z 1385.682,A 0.000,B 0.000,C 90.000,E1 158.773} C_DIS
LIN {X -0.047,Y -466.282,Z 1385.680,A 0.000,B 0.000,C 90.000,E1 158.411} C_DIS
LIN {X 0.090,Y -476.790,Z 1385.675,A 0.000,B 0.000,C 90.000,E1 157.486} C_DIS
LIN {X -0.091,Y -484.010,Z 1385.671,A 0.000,B 0.000,C 90.000,E1 156.847} C_DIS
LIN {X 0.137,Y -494.039,Z 1385.666,A 0.000,B 0.000,C 90.000,E1 155.869} C_DIS
LIN {X -0.022,Y -502.171,Z 1385.661,A 0.000,B 0.000,C 90.000,E1 155.049} C_DIS
LIN {X 0.097,Y -506.060,Z 1385.659,A 0.000,B 0.000,C 90.000,E1 154.613} C_DIS
LIN {X -0.225,Y -513.710,Z 1385.654,A 0.000,B 0.000,C 90.000,E1 153.768} C_DIS
LIN {X 0.066,Y -519.724,Z 1385.650,A 0.000,B 0.000,C 90.000,E1 152.999} C_DIS
LIN {X 0.032,Y -523.108,Z 1385.648,A 0.000,B 0.000,C 90.000,E1 152.564} C_DIS
LIN {X 0.100,Y -527.203,Z 1385.644,A 0.000,B 0.000,C 90.000,E1 151.975} C_DIS
LIN {X 0.202,Y -530.882,Z 1385.641,A 0.000,B 0.000,C 90.000,E1 151.385} C_DIS
LIN {X -0.134,Y -534.178,Z 1385.638,A 0.000,B 0.000,C 90.000,E1 150.845} C_DIS
LIN {X 0.022,Y -537.029,Z 1385.635,A 0.000,B 0.000,C 90.000,E1 150.255} C_DIS
LIN {X -0.081,Y -540.497,Z 1385.630,A 0.000,B 0.000,C 90.000,E1 149.410} C_DIS
LIN {X 0.113,Y -542.629,Z 1385.627,A 0.000,B 0.000,C 90.000,E1 148.820} C_DIS
LIN {X 0.143,Y -544.521,Z 1385.624,A 0.000,B 0.000,C 90.000,E1 148.250} C_DIS
LIN {X 0.105,Y -546.845,Z 1385.619,A 0.000,B 0.000,C 90.000,E1 147.406} C_DIS
LIN {X 0.178,Y -548.184,Z 1385.616,A 0.000,B 0.000,C 90.000,E1 146.834} C_DIS
LIN {X 0.009,Y -549.891,Z 1385.611,A 0.000,B 0.000,C 90.000,E1 146.008} C_DIS
LIN {X -0.142,Y -551.333,Z 1385.607,A 0.000,B 0.000,C 90.000,E1 145.182} C_DIS
LIN {X 0.039,Y -552.531,Z 1385.602,A 0.000,B 0.000,C 90.000,E1 144.322} C_DIS
LIN {X -0.156,Y -553.178,Z 1385.599,A 0.000,B 0.000,C 90.000,E1 143.783} C_DIS
LIN {X 0.046,Y -553.923,Z 1385.594,A 0.000,B 0.000,C 90.000,E1 142.924} C_DIS
LIN {X 0.035,Y -555.248,Z 1385.585,A 0.000,B 0.000,C 90.000,E1 141.251} C_DIS
LIN {X 0.327,Y -556.268,Z 1385.577,A 0.000,B 0.000,C 90.000,E1 139.828} C_DIS
LIN {X 0.125,Y -556.724,Z 1385.572,A 0.000,B 0.000,C 90.000,E1 139.013} C_DIS
LIN {X -0.323,Y -557.464,Z 1385.563,A 0.000,B 0.000,C 90.000,E1 137.391} C_DIS
LIN {X -0.036,Y -558.017,Z 1385.555,A 0.000,B 0.000,C 90.000,E1 135.972} C_DIS
LIN {X 0.314,Y -558.657,Z 1385.546,A 0.000,B 0.000,C 90.000,E1 134.271} C_DIS
LIN {X -0.166,Y -559.109,Z 1385.538,A 0.000,B 0.000,C 90.000,E1 132.933} C_DIS
LIN {X 0.145,Y -559.419,Z 1385.531,A 0.000,B 0.000,C 90.000,E1 131.515} C_DIS
LIN {X -0.279,Y -559.691,Z 1385.523,A 0.000,B 0.000,C 90.000,E1 130.172} C_DIS
LIN {X 0.302,Y -561.016,Z 1385.505,A 0.000,B 0.000,C 90.000,E1 126.790} C_DIS
LIN {X 0.063,Y -561.230,Z 1385.503,A 0.000,B 0.000,C 90.000,E1 126.537} C_DIS
LIN {X -0.149,Y -562.458,Z 1385.500,A 0.000,B 0.000,C 90.000,E1 126.011} C_DIS
LIN {X -0.191,Y -562.503,Z 1385.500,A 0.000,B 0.000,C 90.000,E1 126.011} C_DIS
LIN {X 0.013,Y -564.463,Z 1385.499,A 0.000,B 0.000,C 90.000,E1 125.804} C_DIS
LIN {X 0.121,Y -565.699,Z 1385.499,A 0.000,B 0.000,C 90.000,E1 125.724} C_DIS
LIN {X 0.079,Y -567.938,Z 1385.498,A 0.000,B 0.000,C 90.000,E1 125.644} C_DIS
LIN {X -0.161,Y -578.075,Z 1385.497,A 0.000,B 0.000,C 90.000,E1 125.391} C_DIS
LIN {X 0.092,Y -583.087,Z 1385.496,A 0.000,B 0.000,C 90.000,E1 125.231} C_DIS
LIN {X -0.196,Y -588.746,Z 1385.495,A 0.000,B 0.000,C 90.000,E1 125.025} C_DIS
LIN {X -0.061,Y -591.474,Z 1385.494,A 0.000,B 0.000,C 90.000,E1 124.865} C_DIS
LIN {X -0.056,Y -594.409,Z 1385.493,A 0.000,B 0.000,C 90.000,E1 124.692} C_DIS
LIN {X -0.250,Y -600.184,Z 1385.491,A 0.000,B 0.000,C 90.000,E1 124.326} C_DIS
LIN {X -0.025,Y -604.432,Z 1385.489,A 0.000,B 0.000,C 90.000,E1 123.992} C_DIS
LIN {X -0.367,Y -609.831,Z 1385.486,A 0.000,B 0.000,C 90.000,E1 123.579} C_DIS
LIN {X -0.015,Y -618.862,Z 1385.482,A 0.000,B 0.000,C 90.000,E1 122.704} C_DIS
LIN {X -0.092,Y -624.603,Z 1385.478,A 0.000,B 0.000,C 90.000,E1 122.084} C_DIS
LIN {X 0.232,Y -627.951,Z 1385.476,A 0.000,B 0.000,C 90.000,E1 121.671} C_DIS
LIN {X 0.082,Y -634.952,Z 1385.471,A 0.000,B 0.000,C 90.000,E1 120.797} C_DIS
LIN {X -0.023,Y -640.126,Z 1385.467,A 0.000,B 0.000,C 90.000,E1 120.050} C_DIS
LIN {X 0.093,Y -643.254,Z 1385.464,A 0.000,B 0.000,C 90.000,E1 119.539} C_DIS
LIN {X -0.292,Y -646.449,Z 1385.461,A 0.000,B 0.000,C 90.000,E1 118.949} C_DIS
LIN {X -0.042,Y -649.599,Z 1385.457,A 0.000,B 0.000,C 90.000,E1 118.180} C_DIS
LIN {X -0.031,Y -651.673,Z 1385.453,A 0.000,B 0.000,C 90.000,E1 117.436} C_DIS
LIN {X 0.067,Y -652.026,Z 1385.451,A 0.000,B 0.000,C 90.000,E1 117.180} C_DIS
LIN {X -0.023,Y -652.429,Z 1385.448,A 0.000,B 0.000,C 90.000,E1 116.693} C_DIS
LIN {X 0.189,Y -652.541,Z 1385.446,A 0.000,B 0.000,C 90.000,E1 116.181} C_DIS
LIN {X -0.292,Y -652.418,Z 1385.444,A 0.000,B 0.000,C 90.000,E1 115.976} C_DIS
LIN {X -0.084,Y -651.886,Z 1385.442,A 0.000,B 0.000,C 90.000,E1 115.463} C_DIS
LIN {X 0.120,Y -651.100,Z 1385.439,A 0.000,B 0.000,C 90.000,E1 114.951} C_DIS
LIN {X -0.054,Y -650.496,Z 1385.437,A 0.000,B 0.000,C 90.000,E1 114.719} C_DIS
LIN {X 0.141,Y -648.377,Z 1385.435,A 0.000,B 0.000,C 90.000,E1 114.207} C_DIS
LIN {X 0.232,Y -646.651,Z 1385.433,A 0.000,B 0.000,C 90.000,E1 113.951} C_DIS
LIN {X 0.095,Y -643.516,Z 1385.431,A 0.000,B 0.000,C 90.000,E1 113.590} C_DIS
LIN {X 0.134,Y -641.883,Z 1385.430,A 0.000,B 0.000,C 90.000,E1 113.462} C_DIS
LIN {X 0.075,Y -635.102,Z 1385.428,A 0.000,B 0.000,C 90.000,E1 113.078} C_DIS
LIN {X 0.259,Y -628.479,Z 1385.427,A 0.000,B 0.000,C 90.000,E1 112.823} C_DIS
LIN {X 0.107,Y -617.649,Z 1385.425,A 0.000,B 0.000,C 90.000,E1 112.514} C_DIS
LIN {X 0.115,Y -613.397,Z 1385.424,A 0.000,B 0.000,C 90.000,E1 112.386} C_DIS
LIN {X 0.055,Y -613.272,Z 1385.424,A 0.000,B 0.000,C 90.000,E1 112.386} C_DIS
LIN {X 0.098,Y -624.667,Z 1385.418,A 0.000,B 0.000,C 90.000,E1 111.280} C_DIS
LIN {X 0.073,Y -629.379,Z 1385.416,A 0.000,B 0.000,C 90.000,E1 110.791} C_DIS
LIN {X -0.093,Y -631.621,Z 1385.414,A 0.000,B 0.000,C 90.000,E1 110.556} C_DIS
LIN {X -0.277,Y -635.818,Z 1385.411,A 0.000,B 0.000,C 90.000,E1 110.066} C_DIS
LIN {X 0.182,Y -640.486,Z 1385.408,A 0.000,B 0.000,C 90.000,E1 109.396} C_DIS
LIN {X 0.075,Y -644.554,Z 1385.404,A 0.000,B 0.000,C 90.000,E1 108.779} C_DIS
LIN {X -0.155,Y -649.647,Z 1385.400,A 0.000,B 0.000,C 90.000,E1 107.928} C_DIS
LIN {X 0.061,Y -653.398,Z 1385.395,A 0.000,B 0.000,C 90.000,E1 107.166} C_DIS
LIN {X -0.117,Y -656.343,Z 1385.391,A 0.000,B 0.000,C 90.000,E1 106.441} C_DIS
LIN {X -0.164,Y -657.777,Z 1385.389,A 0.000,B 0.000,C 90.000,E1 105.953} C_DIS
LIN {X 0.250,Y -658.877,Z 1385.386,A 0.000,B 0.000,C 90.000,E1 105.426} C_DIS
LIN {X 0.042,Y -659.804,Z 1385.383,A 0.000,B 0.000,C 90.000,E1 104.954} C_DIS
LIN {X -0.257,Y -660.904,Z 1385.379,A 0.000,B 0.000,C 90.000,E1 104.245} C_DIS
LIN {X 0.098,Y -661.697,Z 1385.375,A 0.000,B 0.000,C 90.000,E1 103.480} C_DIS
LIN {X -0.183,Y -662.014,Z 1385.371,A 0.000,B 0.000,C 90.000,E1 102.771} C_DIS
LIN {X 0.276,Y -661.967,Z 1385.368,A 0.000,B 0.000,C 90.000,E1 102.243} C_DIS
LIN {X 0.087,Y -661.758,Z 1385.365,A 0.000,B 0.000,C 90.000,E1 101.771} C_DIS
LIN {X -0.333,Y -660.994,Z 1385.361,A 0.000,B 0.000,C 90.000,E1 101.074} C_DIS
LIN {X 0.117,Y -660.304,Z 1385.359,A 0.000,B 0.000,C 90.000,E1 100.546} C_DIS
LIN {X -0.312,Y -658.692,Z 1385.355,A 0.000,B 0.000,C 90.000,E1 99.849} C_DIS
LIN {X 0.116,Y -657.447,Z 1385.352,A 0.000,B 0.000,C 90.000,E1 99.321} C_DIS
LIN {X -0.220,Y -655.985,Z 1385.349,A 0.000,B 0.000,C 90.000,E1 98.859} C_DIS
LIN {X 0.086,Y -654.292,Z 1385.346,A 0.000,B 0.000,C 90.000,E1 98.341} C_DIS
LIN {X -0.174,Y -652.392,Z 1385.344,A 0.000,B 0.000,C 90.000,E1 97.871} C_DIS
LIN {X 0.107,Y -650.276,Z 1385.341,A 0.000,B 0.000,C 90.000,E1 97.352} C_DIS
LIN {X 0.259,Y -647.351,Z 1385.338,A 0.000,B 0.000,C 90.000,E1 96.720} C_DIS
LIN {X 0.091,Y -641.898,Z 1385.332,A 0.000,B 0.000,C 90.000,E1 95.739} C_DIS
LIN {X -0.080,Y -636.612,Z 1385.327,A 0.000,B 0.000,C 90.000,E1 94.878} C_DIS
LIN {X 0.219,Y -634.187,Z 1385.325,A 0.000,B 0.000,C 90.000,E1 94.473} C_DIS
LIN {X -0.261,Y -630.651,Z 1385.322,A 0.000,B 0.000,C 90.000,E1 94.012} C_DIS
LIN {X -0.179,Y -626.509,Z 1385.319,A 0.000,B 0.000,C 90.000,E1 93.498} C_DIS
LIN {X -0.085,Y -621.716,Z 1385.317,A 0.000,B 0.000,C 90.000,E1 92.980} C_DIS
LIN {X 0.060,Y -615.171,Z 1385.313,A 0.000,B 0.000,C 90.000,E1 92.350} C_DIS
LIN {X -0.214,Y -608.499,Z 1385.310,A 0.000,B 0.000,C 90.000,E1 91.776} C_DIS
LIN {X 0.265,Y -603.034,Z 1385.307,A 0.000,B 0.000,C 90.000,E1 91.260} C_DIS
LIN {X -0.179,Y -596.941,Z 1385.305,A 0.000,B 0.000,C 90.000,E1 90.859} C_DIS
LIN {X 0.083,Y -593.635,Z 1385.304,A 0.000,B 0.000,C 90.000,E1 90.630} C_DIS
LIN {X 0.139,Y -588.608,Z 1385.302,A 0.000,B 0.000,C 90.000,E1 90.344} C_DIS
LIN {X -0.210,Y -581.651,Z 1385.300,A 0.000,B 0.000,C 90.000,E1 90.057} C_DIS
LIN {X -0.174,Y -578.321,Z 1385.299,A 0.000,B 0.000,C 90.000,E1 89.885} C_DIS
LIN {X 0.202,Y -574.799,Z 1385.298,A 0.000,B 0.000,C 90.000,E1 89.542} C_DIS
LIN {X -0.122,Y -574.393,Z 1385.297,A 0.000,B 0.000,C 90.000,E1 89.542} C_DIS
LIN {X -0.162,Y -574.351,Z 1385.297,A 0.000,B 0.000,C 90.000,E1 89.542} C_DIS
LIN {X -0.087,Y -573.898,Z 1385.297,A 0.000,B 0.000,C 90.000,E1 89.370} C_DIS
LIN {X 0.273,Y -573.731,Z 1385.296,A 0.000,B 0.000,C 90.000,E1 89.198} C_DIS
LIN {X 0.222,Y -573.723,Z 1385.293,A 0.000,B 0.000,C 90.000,E1 88.797} C_DIS
LIN {X -0.044,Y -575.026,Z 1385.284,A 0.000,B 0.000,C 90.000,E1 87.192} C_DIS
LIN {X 0.228,Y -577.268,Z 1385.271,A 0.000,B 0.000,C 90.000,E1 84.723} C_DIS
LIN {X -0.103,Y -579.706,Z 1385.259,A 0.000,B 0.000,C 90.000,E1 82.591} C_DIS
LIN {X -0.230,Y -581.326,Z 1385.251,A 0.000,B 0.000,C 90.000,E1 81.254} C_DIS
LIN {X -0.183,Y -583.246,Z 1385.242,A 0.000,B 0.000,C 90.000,E1 79.634} C_DIS
LIN {X 0.197,Y -584.407,Z 1385.236,A 0.000,B 0.000,C 90.000,E1 78.522} C_DIS
LIN {X -0.054,Y -585.874,Z 1385.227,A 0.000,B 0.000,C 90.000,E1 76.937} C_DIS
LIN {X 0.036,Y -586.998,Z 1385.220,A 0.000,B 0.000,C 90.000,E1 75.589} C_DIS
LIN {X 0.123,Y -588.045,Z 1385.211,A 0.000,B 0.000,C 90.000,E1 73.976} C_DIS
LIN {X 0.238,Y -588.965,Z 1385.202,A 0.000,B 0.000,C 90.000,E1 72.362} C_DIS
LIN {X 0.226,Y -590.043,Z 1385.192,A 0.000,B 0.000,C 90.000,E1 70.496} C_DIS
LIN {X -0.237,Y -590.752,Z 1385.184,A 0.000,B 0.000,C 90.000,E1 69.209} C_DIS
LIN {X 0.083,Y -591.580,Z 1385.177,A 0.000,B 0.000,C 90.000,E1 67.847} C_DIS
LIN {X -0.023,Y -592.900,Z 1385.167,A 0.000,B 0.000,C 90.000,E1 65.997} C_DIS
LIN {X -0.066,Y -594.233,Z 1385.158,A 0.000,B 0.000,C 90.000,E1 64.409} C_DIS
LIN {X 0.103,Y -595.715,Z 1385.148,A 0.000,B 0.000,C 90.000,E1 62.538} C_DIS
LIN {X -0.260,Y -598.241,Z 1385.131,A 0.000,B 0.000,C 90.000,E1 59.665} C_DIS
LIN {X -0.157,Y -599.724,Z 1385.123,A 0.000,B 0.000,C 90.000,E1 58.074} C_DIS
LIN {X -0.219,Y -601.156,Z 1385.114,A 0.000,B 0.000,C 90.000,E1 56.501} C_DIS
LIN {X -0.008,Y -602.837,Z 1385.104,A 0.000,B 0.000,C 90.000,E1 54.642} C_DIS
LIN {X 0.197,Y -604.236,Z 1385.095,A 0.000,B 0.000,C 90.000,E1 53.050} C_DIS
LIN {X -0.084,Y -605.085,Z 1385.089,A 0.000,B 0.000,C 90.000,E1 52.029} C_DIS
LIN {X 0.119,Y -605.799,Z 1385.083,A 0.000,B 0.000,C 90.000,E1 50.964} C_DIS
LIN {X 0.038,Y -606.513,Z 1385.076,A 0.000,B 0.000,C 90.000,E1 49.666} C_DIS
LIN {X -0.020,Y -607.074,Z 1385.069,A 0.000,B 0.000,C 90.000,E1 48.366} C_DIS
LIN {X 0.181,Y -607.334,Z 1385.060,A 0.000,B 0.000,C 90.000,E1 46.782} C_DIS
LIN {X 0.098,Y -607.336,Z 1385.053,A 0.000,B 0.000,C 90.000,E1 45.486} C_DIS
LIN {X 0.021,Y -607.170,Z 1385.046,A 0.000,B 0.000,C 90.000,E1 44.190} C_DIS
LIN {X 0.183,Y -606.567,Z 1385.037,A 0.000,B 0.000,C 90.000,E1 42.609} C_DIS
LIN {X 0.177,Y -605.513,Z 1385.027,A 0.000,B 0.000,C 90.000,E1 40.782} C_DIS
LIN {X 0.088,Y -604.576,Z 1385.019,A 0.000,B 0.000,C 90.000,E1 39.483} C_DIS
LIN {X 0.017,Y -603.916,Z 1385.015,A 0.000,B 0.000,C 90.000,E1 38.705} C_DIS
LIN {X -0.010,Y -602.613,Z 1385.008,A 0.000,B 0.000,C 90.000,E1 37.397} C_DIS
LIN {X -0.067,Y -600.838,Z 1385.000,A 0.000,B 0.000,C 90.000,E1 36.091} C_DIS
LIN {X -0.165,Y -599.520,Z 1384.996,A 0.000,B 0.000,C 90.000,E1 35.311} C_DIS
LIN {X 0.215,Y -597.975,Z 1384.992,A 0.000,B 0.000,C 90.000,E1 34.485} C_DIS
LIN {X -0.019,Y -595.612,Z 1384.986,A 0.000,B 0.000,C 90.000,E1 33.452} C_DIS
LIN {X -0.179,Y -593.649,Z 1384.981,A 0.000,B 0.000,C 90.000,E1 32.673} C_DIS
LIN {X 0.021,Y -590.784,Z 1384.976,A 0.000,B 0.000,C 90.000,E1 31.592} C_DIS
LIN {X 0.104,Y -589.118,Z 1384.973,A 0.000,B 0.000,C 90.000,E1 31.052} C_DIS
LIN {X 0.057,Y -586.148,Z 1384.968,A 0.000,B 0.000,C 90.000,E1 30.256} C_DIS
LIN {X -0.185,Y -584.050,Z 1384.965,A 0.000,B 0.000,C 90.000,E1 29.745} C_DIS
LIN {X -0.280,Y -580.563,Z 1384.961,A 0.000,B 0.000,C 90.000,E1 28.949} C_DIS
LIN {X 0.092,Y -576.753,Z 1384.956,A 0.000,B 0.000,C 90.000,E1 28.103} C_DIS
LIN {X -0.096,Y -572.478,Z 1384.952,A 0.000,B 0.000,C 90.000,E1 27.308} C_DIS
LIN {X -0.082,Y -567.830,Z 1384.947,A 0.000,B 0.000,C 90.000,E1 26.488} C_DIS
LIN {X -0.019,Y -563.736,Z 1384.943,A 0.000,B 0.000,C 90.000,E1 25.796} C_DIS
LIN {X 0.349,Y -560.242,Z 1384.940,A 0.000,B 0.000,C 90.000,E1 25.207} C_DIS
LIN {X 0.343,Y -555.597,Z 1384.936,A 0.000,B 0.000,C 90.000,E1 24.515} C_DIS
LIN {X 0.293,Y -550.628,Z 1384.933,A 0.000,B 0.000,C 90.000,E1 23.823} C_DIS
LIN {X -0.013,Y -545.102,Z 1384.929,A 0.000,B 0.000,C 90.000,E1 23.153} C_DIS
LIN {X -0.145,Y -538.277,Z 1384.924,A 0.000,B 0.000,C 90.000,E1 22.333} C_DIS
LIN {X -0.202,Y -533.302,Z 1384.921,A 0.000,B 0.000,C 90.000,E1 21.770} C_DIS
LIN {X 0.069,Y -523.083,Z 1384.915,A 0.000,B 0.000,C 90.000,E1 20.610} C_DIS
LIN {X -0.142,Y -512.366,Z 1384.908,A 0.000,B 0.000,C 90.000,E1 19.504} C_DIS
LIN {X -0.153,Y -501.718,Z 1384.902,A 0.000,B 0.000,C 90.000,E1 18.417} C_DIS
LIN {X -0.117,Y -485.098,Z 1384.893,A 0.000,B 0.000,C 90.000,E1 16.732} C_DIS
LIN {X -0.167,Y -470.019,Z 1384.884,A 0.000,B 0.000,C 90.000,E1 15.190} C_DIS
LIN {X -0.130,Y -460.212,Z 1384.879,A 0.000,B 0.000,C 90.000,E1 14.175} C_DIS
LIN {X -0.196,Y -447.776,Z 1384.871,A 0.000,B 0.000,C 90.000,E1 12.883} C_DIS
LIN {X -0.176,Y -427.070,Z 1384.859,A 0.000,B 0.000,C 90.000,E1 10.602} C_DIS
LIN {X -0.057,Y -412.079,Z 1384.849,A 0.000,B 0.000,C 90.000,E1 8.803} C_DIS
LIN {X 0.050,Y -399.716,Z 1384.841,A 0.000,B 0.000,C 90.000,E1 7.296} C_DIS
LIN {X 0.194,Y -393.485,Z 1384.836,A 0.000,B 0.000,C 90.000,E1 6.486} C_DIS
LIN {X 0.157,Y -392.269,Z 1384.835,A 0.000,B 0.000,C 90.000,E1 6.315} C_DIS
LIN {X -0.036,Y -390.507,Z 1384.833,A 0.000,B 0.000,C 90.000,E1 6.030} C_DIS
LIN {X -0.073,Y -390.495,Z 1384.833,A 0.000,B 0.000,C 90.000,E1 6.030} C_DIS
LIN {X 0.130,Y -390.464,Z 1384.833,A 0.000,B 0.000,C 90.000,E1 5.967} C_DIS
LIN {X 0.092,Y -390.478,Z 1384.833,A 0.000,B 0.000,C 90.000,E1 5.967} C_DIS
LIN {X 0.163,Y -393.391,Z 1384.831,A 0.000,B 0.000,C 90.000,E1 5.568} C_DIS
LIN {X -0.091,Y -398.995,Z 1384.828,A 0.000,B 0.000,C 90.000,E1 5.106} C_DIS
LIN {X -0.037,Y -403.414,Z 1384.826,A 0.000,B 0.000,C 90.000,E1 4.759} C_DIS
LIN {X 0.139,Y -410.920,Z 1384.823,A 0.000,B 0.000,C 90.000,E1 4.073} C_DIS
LIN {X 0.017,Y -416.644,Z 1384.819,A 0.000,B 0.000,C 90.000,E1 3.498} C_DIS
LIN {X 0.014,Y -423.234,Z 1384.815,A 0.000,B 0.000,C 90.000,E1 2.694} C_DIS
LIN {X 0.203,Y -430.512,Z 1384.809,A 0.000,B 0.000,C 90.000,E1 1.661} C_DIS
LIN {X -0.032,Y -436.287,Z 1384.805,A 0.000,B 0.000,C 90.000,E1 0.859} C_DIS
LIN {X 0.000,Y -441.888,Z 1384.800,A 0.000,B 0.000,C 90.000,E1 360.000} C_DIS
LIN {X -0.017,Y -447.301,Z 1384.795,A 0.000,B 0.000,C 90.000,E1 359.141} C_DIS
LIN {X -0.095,Y -452.073,Z 1384.791,A 0.000,B 0.000,C 90.000,E1 358.339} C_DIS
LIN {X -0.116,Y -456.484,Z 1384.786,A 0.000,B 0.000,C 90.000,E1 357.535} C_DIS
LIN {X -0.087,Y -460.588,Z 1384.782,A 0.000,B 0.000,C 90.000,E1 356.731} C_DIS
LIN {X -0.151,Y -463.681,Z 1384.778,A 0.000,B 0.000,C 90.000,E1 356.102} C_DIS
LIN {X -0.055,Y -467.232,Z 1384.774,A 0.000,B 0.000,C 90.000,E1 355.298} C_DIS
LIN {X 0.235,Y -471.129,Z 1384.769,A 0.000,B 0.000,C 90.000,E1 354.318} C_DIS
LIN {X -0.186,Y -473.563,Z 1384.765,A 0.000,B 0.000,C 90.000,E1 353.742} C_DIS
LIN {X 0.013,Y -478.042,Z 1384.758,A 0.000,B 0.000,C 90.000,E1 352.470} C_DIS
LIN {X 0.106,Y -479.819,Z 1384.755,A 0.000,B 0.000,C 90.000,E1 351.837} C_DIS
LIN {X -0.045,Y -480.423,Z 1384.753,A 0.000,B 0.000,C 90.000,E1 351.546} C_DIS
LIN {X -0.192,Y -480.789,Z 1384.751,A 0.000,B 0.000,C 90.000,E1 351.254} C_DIS
LIN {X 0.139,Y -480.800,Z 1384.750,A 0.000,B 0.000,C 90.000,E1 350.905} C_DIS
LIN {X -0.082,Y -480.087,Z 1384.748,A 0.000,B 0.000,C 90.000,E1 350.622} C_DIS
LIN {X -0.127,Y -479.098,Z 1384.747,A 0.000,B 0.000,C 90.000,E1 350.500} C_DIS
LIN {X 0.060,Y -475.860,Z 1384.747,A 0.000,B 0.000,C 90.000,E1 350.387} C_DIS
LIN {X -0.015,Y -435.377,Z 1384.742,A 0.000,B 0.000,C 90.000,E1 349.511} C_DIS
LIN {X 0.014,Y -399.696,Z 1384.737,A 0.000,B 0.000,C 90.000,E1 348.578} C_DIS
LIN {X 0.046,Y -367.789,Z 1384.731,A 0.000,B 0.000,C 90.000,E1 347.589} C_DIS
LIN {X 0.070,Y -359.390,Z 1384.729,A 0.000,B 0.000,C 90.000,E1 347.297} C_DIS
LIN {X 0.046,Y -359.289,Z 1384.729,A 0.000,B 0.000,C 90.000,E1 347.297} C_DIS
LIN {X 0.095,Y -359.583,Z 1384.725,A 0.000,B 0.000,C 90.000,E1 346.464} C_DIS
LIN {X 0.124,Y -361.919,Z 1384.683,A 0.000,B 0.000,C 90.000,E1 338.954} C_DIS
LIN {X -0.018,Y -366.136,Z 1384.642,A 0.000,B 0.000,C 90.000,E1 331.513} C_DIS
LIN {X -0.011,Y -371.113,Z 1384.605,A 0.000,B 0.000,C 90.000,E1 324.848} C_DIS
LIN {X -0.035,Y -371.854,Z 1384.601,A 0.000,B 0.000,C 90.000,E1 324.116} C_DIS
LIN {X 0.043,Y -377.560,Z 1384.566,A 0.000,B 0.000,C 90.000,E1 317.877} C_DIS
LIN {X 0.031,Y -378.042,Z 1384.564,A 0.000,B 0.000,C 90.000,E1 317.514} C_DIS
LIN {X 0.037,Y -383.666,Z 1384.532,A 0.000,B 0.000,C 90.000,E1 311.714} C_DIS
LIN {X 0.086,Y -384.652,Z 1384.528,A 0.000,B 0.000,C 90.000,E1 310.987} C_DIS
LIN {X -0.115,Y -385.239,Z 1384.524,A 0.000,B 0.000,C 90.000,E1 310.297} C_DIS
LIN {X 0.145,Y -391.299,Z 1384.492,A 0.000,B 0.000,C 90.000,E1 304.532} C_DIS
LIN {X -0.058,Y -397.011,Z 1384.458,A 0.000,B 0.000,C 90.000,E1 298.537} C_DIS
LIN {X 0.073,Y -401.379,Z 1384.427,A 0.000,B 0.000,C 90.000,E1 292.898} C_DIS
LIN {X -0.217,Y -401.663,Z 1384.425,A 0.000,B 0.000,C 90.000,E1 292.589} C_DIS
LIN {X -0.064,Y -404.757,Z 1384.394,A 0.000,B 0.000,C 90.000,E1 286.985} C_DIS
LIN {X -0.051,Y -406.158,Z 1384.364,A 0.000,B 0.000,C 90.000,E1 281.422} C_DIS
LIN {X 0.052,Y -405.665,Z 1384.333,A 0.000,B 0.000,C 90.000,E1 275.853} C_DIS
LIN {X 0.124,Y -403.561,Z 1384.306,A 0.000,B 0.000,C 90.000,E1 270.974} C_DIS
LIN {X 0.059,Y -403.144,Z 1384.302,A 0.000,B 0.000,C 90.000,E1 270.286} C_DIS
LIN {X -0.110,Y -399.052,Z 1384.273,A 0.000,B 0.000,C 90.000,E1 265.065} C_DIS
LIN {X -0.168,Y -398.729,Z 1384.271,A 0.000,B 0.000,C 90.000,E1 264.723} C_DIS
LIN {X 0.110,Y -393.265,Z 1384.243,A 0.000,B 0.000,C 90.000,E1 259.746} C_DIS
LIN {X 0.030,Y -392.615,Z 1384.239,A 0.000,B 0.000,C 90.000,E1 259.050} C_DIS
LIN {X 0.188,Y -386.211,Z 1384.214,A 0.000,B 0.000,C 90.000,E1 254.393} C_DIS
LIN {X 0.151,Y -385.111,Z 1384.208,A 0.000,B 0.000,C 90.000,E1 253.323} C_DIS
LIN {X 0.029,Y -377.772,Z 1384.181,A 0.000,B 0.000,C 90.000,E1 248.646} C_DIS
LIN {X 0.110,Y -376.033,Z 1384.173,A 0.000,B 0.000,C 90.000,E1 247.177} C_DIS
LIN {X -0.110,Y -369.224,Z 1384.151,A 0.000,B 0.000,C 90.000,E1 243.179} C_DIS
LIN {X 0.127,Y -366.358,Z 1384.139,A 0.000,B 0.000,C 90.000,E1 240.923} C_DIS
LIN {X 0.049,Y -364.353,Z 1384.132,A 0.000,B 0.000,C 90.000,E1 239.822} C_DIS
LIN {X -0.016,Y -357.479,Z 1384.108,A 0.000,B 0.000,C 90.000,E1 235.341} C_DIS
LIN {X 0.073,Y -356.139,Z 1384.101,A 0.000,B 0.000,C 90.000,E1 234.196} C_DIS
LIN {X 0.148,Y -354.213,Z 1384.095,A 0.000,B 0.000,C 90.000,E1 233.050} C_DIS
LIN {X 0.098,Y -347.664,Z 1384.069,A 0.000,B 0.000,C 90.000,E1 228.485} C_DIS
LIN {X -0.120,Y -346.016,Z 1384.061,A 0.000,B 0.000,C 90.000,E1 226.986} C_DIS
LIN {X 0.105,Y -339.216,Z 1384.033,A 0.000,B 0.000,C 90.000,E1 221.919} C_DIS
LIN {X 0.192,Y -337.028,Z 1384.020,A 0.000,B 0.000,C 90.000,E1 219.564} C_DIS
LIN {X -0.094,Y -336.088,Z 1384.016,A 0.000,B 0.000,C 90.000,E1 218.830} C_DIS
LIN {X 0.048,Y -330.435,Z 1383.985,A 0.000,B 0.000,C 90.000,E1 213.293} C_DIS
LIN {X -0.100,Y -329.163,Z 1383.974,A 0.000,B 0.000,C 90.000,E1 211.337} C_DIS
LIN {X -0.065,Y -324.417,Z 1383.939,A 0.000,B 0.000,C 90.000,E1 204.951} C_DIS
LIN {X -0.081,Y -323.735,Z 1383.927,A 0.000,B 0.000,C 90.000,E1 202.950} C_DIS
LIN {X -0.173,Y -321.121,Z 1383.882,A 0.000,B 0.000,C 90.000,E1 194.717} C_DIS
LIN {X 0.119,Y -321.178,Z 1383.882,A 0.000,B 0.000,C 90.000,E1 194.662} C_DIS
LIN {X -0.044,Y -347.450,Z 1383.875,A 0.000,B 0.000,C 90.000,E1 193.592} C_DIS
LIN {X 0.034,Y -376.722,Z 1383.870,A 0.000,B 0.000,C 90.000,E1 192.535} C_DIS
LIN {X 0.033,Y -409.798,Z 1383.864,A 0.000,B 0.000,C 90.000,E1 191.535} C_DIS
LIN {X 0.197,Y -435.566,Z 1383.860,A 0.000,B 0.000,C 90.000,E1 190.838} C_DIS
LIN {X -0.067,Y -436.850,Z 1383.860,A 0.000,B 0.000,C 90.000,E1 190.782} C_DIS
LIN {X -0.022,Y -438.054,Z 1383.859,A 0.000,B 0.000,C 90.000,E1 190.546} C_DIS
LIN {X 0.118,Y -438.803,Z 1383.857,A 0.000,B 0.000,C 90.000,E1 190.197} C_DIS
LIN {X -0.170,Y -439.094,Z 1383.855,A 0.000,B 0.000,C 90.000,E1 189.905} C_DIS
LIN {X 0.127,Y -439.090,Z 1383.851,A 0.000,B 0.000,C 90.000,E1 189.208} C_DIS
LIN {X -0.210,Y -438.773,Z 1383.844,A 0.000,B 0.000,C 90.000,E1 187.936} C_DIS
LIN {X -0.115,Y -438.409,Z 1383.837,A 0.000,B 0.000,C 90.000,E1 186.606} C_DIS
LIN {X -0.032,Y -437.990,Z 1383.829,A 0.000,B 0.000,C 90.000,E1 185.277} C_DIS
LIN {X -0.136,Y -437.366,Z 1383.824,A 0.000,B 0.000,C 90.000,E1 184.302} C_DIS
LIN {X 0.093,Y -436.831,Z 1383.820,A 0.000,B 0.000,C 90.000,E1 183.612} C_DIS
LIN {X 0.075,Y -435.111,Z 1383.813,A 0.000,B 0.000,C 90.000,E1 182.293} C_DIS
LIN {X -0.062,Y -433.620,Z 1383.807,A 0.000,B 0.000,C 90.000,E1 181.318} C_DIS
LIN {X 0.204,Y -431.821,Z 1383.802,A 0.000,B 0.000,C 90.000,E1 180.286} C_DIS
LIN {X -0.060,Y -430.287,Z 1383.798,A 0.000,B 0.000,C 90.000,E1 179.656} C_DIS
LIN {X 0.164,Y -427.542,Z 1383.792,A 0.000,B 0.000,C 90.000,E1 178.625} C_DIS
LIN {X -0.061,Y -424.307,Z 1383.787,A 0.000,B 0.000,C 90.000,E1 177.650} C_DIS
LIN {X 0.080,Y -420.961,Z 1383.782,A 0.000,B 0.000,C 90.000,E1 176.788} C_DIS
LIN {X 0.145,Y -417.904,Z 1383.779,A 0.000,B 0.000,C 90.000,E1 176.102} C_DIS
LIN {X -0.163,Y -412.530,Z 1383.773,A 0.000,B 0.000,C 90.000,E1 175.122} C_DIS
LIN {X -0.157,Y -406.142,Z 1383.767,A 0.000,B 0.000,C 90.000,E1 174.090} C_DIS
LIN {X 0.093,Y -390.243,Z 1383.753,A 0.000,B 0.000,C 90.000,E1 171.602} C_DIS
LIN {X 0.152,Y -380.068,Z 1383.744,A 0.000,B 0.000,C 90.000,E1 169.803} C_DIS
LIN {X -0.045,Y -375.415,Z 1383.739,A 0.000,B 0.000,C 90.000,E1 168.926} C_DIS
LIN {X -0.138,Y -373.097,Z 1383.735,A 0.000,B 0.000,C 90.000,E1 168.398} C_DIS
LIN {X 0.110,Y -371.706,Z 1383.733,A 0.000,B 0.000,C 90.000,E1 167.993} C_DIS
LIN {X 0.070,Y -370.963,Z 1383.731,A 0.000,B 0.000,C 90.000,E1 167.645} C_DIS
LIN {X -0.121,Y -370.983,Z 1383.731,A 0.000,B 0.000,C 90.000,E1 167.589} C_DIS
LIN {X -0.112,Y -372.079,Z 1383.728,A 0.000,B 0.000,C 90.000,E1 167.117} C_DIS
LIN {X -0.150,Y -372.101,Z 1383.728,A 0.000,B 0.000,C 90.000,E1 167.117} C_DIS
LIN {X -0.152,Y -375.383,Z 1383.725,A 0.000,B 0.000,C 90.000,E1 166.589} C_DIS
LIN {X 0.146,Y -381.006,Z 1383.721,A 0.000,B 0.000,C 90.000,E1 165.825} C_DIS
LIN {X 0.099,Y -392.716,Z 1383.714,A 0.000,B 0.000,C 90.000,E1 164.574} C_DIS
LIN {X 0.119,Y -405.059,Z 1383.708,A 0.000,B 0.000,C 90.000,E1 163.378} C_DIS
LIN {X 0.176,Y -419.189,Z 1383.701,A 0.000,B 0.000,C 90.000,E1 162.127} C_DIS
LIN {X 0.125,Y -441.179,Z 1383.691,A 0.000,B 0.000,C 90.000,E1 160.369} C_DIS
LIN {X 0.228,Y -453.597,Z 1383.686,A 0.000,B 0.000,C 90.000,E1 159.390} C_DIS
LIN {X 0.242,Y -461.348,Z 1383.682,A 0.000,B 0.000,C 90.000,E1 158.773} C_DIS
LIN {X 0.142,Y -467.415,Z 1383.679,A 0.000,B 0.000,C 90.000,E1 158.284} C_DIS
LIN {X -0.100,Y -476.395,Z 1383.675,A 0.000,B 0.000,C 90.000,E1 157.539} C_DIS
LIN {X -0.009,Y -483.631,Z 1383.672,A 0.000,B 0.000,C 90.000,E1 156.869} C_DIS
LIN {X -0.011,Y -493.633,Z 1383.666,A 0.000,B 0.000,C 90.000,E1 155.921} C_DIS
LIN {X -0.165,Y -501.786,Z 1383.662,A 0.000,B 0.000,C 90.000,E1 155.101} C_DIS
LIN {X -0.061,Y -505.722,Z 1383.659,A 0.000,B 0.000,C 90.000,E1 154.665} C_DIS
LIN {X 0.069,Y -513.391,Z 1383.654,A 0.000,B 0.000,C 90.000,E1 153.768} C_DIS
LIN {X -0.086,Y -519.417,Z 1383.650,A 0.000,B 0.000,C 90.000,E1 153.050} C_DIS
LIN {X -0.122,Y -522.828,Z 1383.648,A 0.000,B 0.000,C 90.000,E1 152.615} C_DIS
LIN {X -0.046,Y -526.981,Z 1383.645,A 0.000,B 0.000,C 90.000,E1 152.025} C_DIS
LIN {X 0.055,Y -530.685,Z 1383.641,A 0.000,B 0.000,C 90.000,E1 151.435} C_DIS
LIN {X 0.187,Y -533.968,Z 1383.638,A 0.000,B 0.000,C 90.000,E1 150.845} C_DIS
LIN {X 0.202,Y -537.430,Z 1383.634,A 0.000,B 0.000,C 90.000,E1 150.127} C_DIS
LIN {X -0.034,Y -541.421,Z 1383.629,A 0.000,B 0.000,C 90.000,E1 149.154} C_DIS
LIN {X -0.283,Y -544.347,Z 1383.624,A 0.000,B 0.000,C 90.000,E1 148.329} C_DIS
LIN {X -0.034,Y -546.675,Z 1383.619,A 0.000,B 0.000,C 90.000,E1 147.454} C_DIS
LIN {X -0.260,Y -548.024,Z 1383.616,A 0.000,B 0.000,C 90.000,E1 146.914} C_DIS
LIN {X 0.330,Y -549.744,Z 1383.611,A 0.000,B 0.000,C 90.000,E1 146.008} C_DIS
LIN {X 0.178,Y -551.197,Z 1383.607,A 0.000,B 0.000,C 90.000,E1 145.182} C_DIS
LIN {X 0.099,Y -552.752,Z 1383.600,A 0.000,B 0.000,C 90.000,E1 144.069} C_DIS
LIN {X -0.148,Y -553.588,Z 1383.596,A 0.000,B 0.000,C 90.000,E1 143.256} C_DIS
LIN {X 0.206,Y -554.683,Z 1383.588,A 0.000,B 0.000,C 90.000,E1 141.823} C_DIS
LIN {X 0.137,Y -555.711,Z 1383.580,A 0.000,B 0.000,C 90.000,E1 140.436} C_DIS
LIN {X 0.001,Y -556.433,Z 1383.574,A 0.000,B 0.000,C 90.000,E1 139.337} C_DIS
LIN {X -0.084,Y -557.220,Z 1383.565,A 0.000,B 0.000,C 90.000,E1 137.676} C_DIS
LIN {X -0.181,Y -557.786,Z 1383.557,A 0.000,B 0.000,C 90.000,E1 136.296} C_DIS
LIN {X 0.165,Y -558.418,Z 1383.548,A 0.000,B 0.000,C 90.000,E1 134.595} C_DIS
LIN {X 0.064,Y -558.895,Z 1383.540,A 0.000,B 0.000,C 90.000,E1 133.218} C_DIS
LIN {X -0.006,Y -559.258,Z 1383.532,A 0.000,B 0.000,C 90.000,E1 131.838} C_DIS
LIN {X -0.067,Y -559.535,Z 1383.525,A 0.000,B 0.000,C 90.000,E1 130.458} C_DIS
LIN {X -0.026,Y -560.566,Z 1383.509,A 0.000,B 0.000,C 90.000,E1 127.684} C_DIS
LIN {X 0.069,Y -560.838,Z 1383.508,A 0.000,B 0.000,C 90.000,E1 127.397} C_DIS
LIN {X -0.185,Y -561.274,Z 1383.505,A 0.000,B 0.000,C 90.000,E1 126.870} C_DIS
LIN {X -0.320,Y -561.685,Z 1383.504,A 0.000,B 0.000,C 90.000,E1 126.664} C_DIS
LIN {X 0.117,Y -562.682,Z 1383.502,A 0.000,B 0.000,C 90.000,E1 126.377} C_DIS
LIN {X 0.074,Y -562.747,Z 1383.502,A 0.000,B 0.000,C 90.000,E1 126.377} C_DIS
LIN {X 0.181,Y -566.425,Z 1383.501,A 0.000,B 0.000,C 90.000,E1 126.171} C_DIS
LIN {X 0.107,Y -567.740,Z 1383.501,A 0.000,B 0.000,C 90.000,E1 126.091} C_DIS
LIN {X 0.147,Y -577.948,Z 1383.499,A 0.000,B 0.000,C 90.000,E1 125.804} C_DIS
LIN {X 0.138,Y -584.482,Z 1383.498,A 0.000,B 0.000,C 90.000,E1 125.598} C_DIS
LIN {X 0.014,Y -586.842,Z 1383.497,A 0.000,B 0.000,C 90.000,E1 125.518} C_DIS
LIN {X -0.060,Y -589.635,Z 1383.497,A 0.000,B 0.000,C 90.000,E1 125.391} C_DIS
LIN {X -0.042,Y -592.579,Z 1383.496,A 0.000,B 0.000,C 90.000,E1 125.231} C_DIS
LIN {X 0.129,Y -596.887,Z 1383.494,A 0.000,B 0.000,C 90.000,E1 124.945} C_DIS
LIN {X 0.192,Y -602.686,Z 1383.492,A 0.000,B 0.000,C 90.000,E1 124.532} C_DIS
LIN {X -0.075,Y -608.127,Z 1383.490,A 0.000,B 0.000,C 90.000,E1 124.119} C_DIS
LIN {X 0.307,Y -615.931,Z 1383.486,A 0.000,B 0.000,C 90.000,E1 123.372} C_DIS
LIN {X 0.339,Y -620.983,Z 1383.483,A 0.000,B 0.000,C 90.000,E1 122.880} C_DIS
LIN {X -0.073,Y -626.613,Z 1383.479,A 0.000,B 0.000,C 90.000,E1 122.291} C_DIS
LIN {X 0.266,Y -629.839,Z 1383.477,A 0.000,B 0.000,C 90.000,E1 121.878} C_DIS
LIN {X 0.093,Y -633.888,Z 1383.474,A 0.000,B 0.000,C 90.000,E1 121.386} C_DIS
LIN {X 0.158,Y -637.661,Z 1383.472,A 0.000,B 0.000,C 90.000,E1 120.875} C_DIS
LIN {X 0.028,Y -641.207,Z 1383.469,A 0.000,B 0.000,C 90.000,E1 120.384} C_DIS
LIN {X 0.183,Y -645.003,Z 1383.465,A 0.000,B 0.000,C 90.000,E1 119.745} C_DIS
LIN {X -0.227,Y -647.603,Z 1383.463,A 0.000,B 0.000,C 90.000,E1 119.283} C_DIS
LIN {X 0.347,Y -650.984,Z 1383.458,A 0.000,B 0.000,C 90.000,E1 118.487} C_DIS
LIN {X 0.067,Y -653.267,Z 1383.454,A 0.000,B 0.000,C 90.000,E1 117.769} C_DIS
LIN {X 0.172,Y -653.780,Z 1383.453,A 0.000,B 0.000,C 90.000,E1 117.513} C_DIS
LIN {X -0.194,Y -654.344,Z 1383.450,A 0.000,B 0.000,C 90.000,E1 117.052} C_DIS
LIN {X 0.025,Y -654.733,Z 1383.448,A 0.000,B 0.000,C 90.000,E1 116.539} C_DIS
LIN {X -0.041,Y -654.514,Z 1383.445,A 0.000,B 0.000,C 90.000,E1 116.052} C_DIS
LIN {X -0.294,Y -653.824,Z 1383.441,A 0.000,B 0.000,C 90.000,E1 115.335} C_DIS
LIN {X -0.078,Y -653.041,Z 1383.438,A 0.000,B 0.000,C 90.000,E1 114.823} C_DIS
LIN {X -0.244,Y -652.188,Z 1383.437,A 0.000,B 0.000,C 90.000,E1 114.591} C_DIS
LIN {X -0.037,Y -649.891,Z 1383.434,A 0.000,B 0.000,C 90.000,E1 114.079} C_DIS
LIN {X 0.146,Y -645.621,Z 1383.431,A 0.000,B 0.000,C 90.000,E1 113.567} C_DIS
LIN {X -0.071,Y -644.279,Z 1383.430,A 0.000,B 0.000,C 90.000,E1 113.462} C_DIS
LIN {X -0.172,Y -640.552,Z 1383.429,A 0.000,B 0.000,C 90.000,E1 113.259} C_DIS
LIN {X -0.101,Y -635.807,Z 1383.428,A 0.000,B 0.000,C 90.000,E1 113.003} C_DIS
LIN {X -0.068,Y -629.180,Z 1383.427,A 0.000,B 0.000,C 90.000,E1 112.770} C_DIS
LIN {X -0.088,Y -618.390,Z 1383.425,A 0.000,B 0.000,C 90.000,E1 112.461} C_DIS
LIN {X 0.303,Y -615.266,Z 1383.424,A 0.000,B 0.000,C 90.000,E1 112.333} C_DIS
LIN {X 0.251,Y -615.305,Z 1383.424,A 0.000,B 0.000,C 90.000,E1 112.333} C_DIS
LIN {X -0.030,Y -624.946,Z 1383.419,A 0.000,B 0.000,C 90.000,E1 111.408} C_DIS
LIN {X -0.139,Y -628.536,Z 1383.417,A 0.000,B 0.000,C 90.000,E1 111.046} C_DIS
LIN {X -0.034,Y -631.960,Z 1383.415,A 0.000,B 0.000,C 90.000,E1 110.663} C_DIS
LIN {X -0.221,Y -636.172,Z 1383.412,A 0.000,B 0.000,C 90.000,E1 110.174} C_DIS
LIN {X 0.024,Y -640.831,Z 1383.409,A 0.000,B 0.000,C 90.000,E1 109.523} C_DIS
LIN {X -0.055,Y -645.585,Z 1383.404,A 0.000,B 0.000,C 90.000,E1 108.779} C_DIS
LIN {X 0.344,Y -650.615,Z 1383.400,A 0.000,B 0.000,C 90.000,E1 107.873} C_DIS
LIN {X -0.051,Y -654.345,Z 1383.395,A 0.000,B 0.000,C 90.000,E1 107.166} C_DIS
LIN {X -0.219,Y -657.288,Z 1383.391,A 0.000,B 0.000,C 90.000,E1 106.441} C_DIS
LIN {X 0.373,Y -658.733,Z 1383.389,A 0.000,B 0.000,C 90.000,E1 105.898} C_DIS
LIN {X 0.161,Y -659.847,Z 1383.386,A 0.000,B 0.000,C 90.000,E1 105.426} C_DIS
LIN {X -0.042,Y -660.792,Z 1383.383,A 0.000,B 0.000,C 90.000,E1 104.954} C_DIS
LIN {X -0.331,Y -661.911,Z 1383.379,A 0.000,B 0.000,C 90.000,E1 104.245} C_DIS
LIN {X 0.125,Y -662.468,Z 1383.376,A 0.000,B 0.000,C 90.000,E1 103.716} C_DIS
LIN {X -0.057,Y -662.852,Z 1383.374,A 0.000,B 0.000,C 90.000,E1 103.244} C_DIS
LIN {X -0.238,Y -663.031,Z 1383.371,A 0.000,B 0.000,C 90.000,E1 102.771} C_DIS
LIN {X 0.229,Y -662.997,Z 1383.368,A 0.000,B 0.000,C 90.000,E1 102.243} C_DIS
LIN {X 0.046,Y -662.786,Z 1383.365,A 0.000,B 0.000,C 90.000,E1 101.771} C_DIS
LIN {X -0.364,Y -662.004,Z 1383.361,A 0.000,B 0.000,C 90.000,E1 101.074} C_DIS
LIN {X 0.094,Y -661.336,Z 1383.359,A 0.000,B 0.000,C 90.000,E1 100.546} C_DIS
LIN {X -0.327,Y -659.735,Z 1383.355,A 0.000,B 0.000,C 90.000,E1 99.849} C_DIS
LIN {X 0.110,Y -658.474,Z 1383.352,A 0.000,B 0.000,C 90.000,E1 99.321} C_DIS
LIN {X -0.221,Y -657.019,Z 1383.349,A 0.000,B 0.000,C 90.000,E1 98.859} C_DIS
LIN {X 0.092,Y -655.347,Z 1383.346,A 0.000,B 0.000,C 90.000,E1 98.341} C_DIS
LIN {X -0.161,Y -653.436,Z 1383.344,A 0.000,B 0.000,C 90.000,E1 97.871} C_DIS
LIN {X 0.128,Y -651.322,Z 1383.341,A 0.000,B 0.000,C 90.000,E1 97.352} C_DIS
LIN {X 0.288,Y -648.419,Z 1383.338,A 0.000,B 0.000,C 90.000,E1 96.720} C_DIS
LIN {X 0.133,Y -642.940,Z 1383.332,A 0.000,B 0.000,C 90.000,E1 95.739} C_DIS
LIN {X -0.026,Y -637.656,Z 1383.327,A 0.000,B 0.000,C 90.000,E1 94.878} C_DIS
LIN {X 0.279,Y -635.262,Z 1383.325,A 0.000,B 0.000,C 90.000,E1 94.473} C_DIS
LIN {X -0.196,Y -631.775,Z 1383.322,A 0.000,B 0.000,C 90.000,E1 94.012} C_DIS
LIN {X -0.106,Y -627.663,Z 1383.319,A 0.000,B 0.000,C 90.000,E1 93.498} C_DIS
LIN {X -0.148,Y -621.705,Z 1383.316,A 0.000,B 0.000,C 90.000,E1 92.865} C_DIS
LIN {X -0.082,Y -613.754,Z 1383.312,A 0.000,B 0.000,C 90.000,E1 92.121} C_DIS
LIN {X -0.265,Y -608.448,Z 1383.309,A 0.000,B 0.000,C 90.000,E1 91.661} C_DIS
LIN {X 0.236,Y -602.990,Z 1383.307,A 0.000,B 0.000,C 90.000,E1 91.146} C_DIS
LIN {X -0.166,Y -596.813,Z 1383.304,A 0.000,B 0.000,C 90.000,E1 90.745} C_DIS
LIN {X -0.073,Y -590.037,Z 1383.302,A 0.000,B 0.000,C 90.000,E1 90.344} C_DIS
LIN {X 0.071,Y -582.785,Z 1383.300,A 0.000,B 0.000,C 90.000,E1 90.000} C_DIS
LIN {X -0.249,Y -578.833,Z 1383.299,A 0.000,B 0.000,C 90.000,E1 89.828} C_DIS
LIN {X -0.173,Y -576.545,Z 1383.298,A 0.000,B 0.000,C 90.000,E1 89.656} C_DIS
LIN {X 0.060,Y -574.677,Z 1383.297,A 0.000,B 0.000,C 90.000,E1 89.484} C_DIS
LIN {X 0.025,Y -574.646,Z 1383.297,A 0.000,B 0.000,C 90.000,E1 89.484} C_DIS
